(* rising edge trigger *)
IF in AND NOT edge THEN
	start := Tx;
	IF pt > t#0ms THEN Q := TRUE; END_IF;
END_IF;
edge := in;
IF q THEN
	et := Tx - start;
	IF et >= PT THEN
		Q := FALSE;
		et := t#0ms;
	END_IF;
END_IF;


(* revision history
hm	4. aug 2006		rev 1.0
	original version

hm	17. sep 2007	rev 1.1
	replaced time() with T_PLC_MS() for compatibility reasons
	
*)
END_FUNCTION_BLOCK

(* POU engineering/signal generators/pwm_pw, ST *)
FUNCTION_BLOCK pwm_pw
VAR_INPUT
	F : REAL;
	PW : TIME;
END_VAR
VAR_OUTPUT
	Q : BOOL;
END_VAR
VAR
	clk: CLK_Prg;
	pulse: TP_R;
END_VAR

(*
	version 1.1	25 feb 2007
	programmer 	oscat
	tested BY		oscat

this signal generator generates a square wave signal which is specified by the frequency and the pulse width.
*)
CLK(PT := REAL_TO_TIME(1000/F));
Pulse(in := clk.Q, pt := pw);
Q := pulse.Q;

(* revision history

hm		25. feb 2007	rev 1.1
	recoded in st for better performance and better portability

*)
END_FUNCTION_BLOCK

(* POU engineering/signal generators/rmp_soft, ST *)
FUNCTION_BLOCK rmp_soft
VAR_INPUT
	IN : BOOL;
	val : BYTE;
END_VAR
VAR_INPUT CONSTANT
	pt_on: TIME := T#100ms;
	PT_off : TIME := T#100ms;
END_VAR
VAR CONSTANT
	steps : INT := 255;
END_VAR
VAR_OUTPUT
	Out : BYTE := 0;
END_VAR
VAR
	last_step : TIME := T#0ms;
	now : TIME;
	x :REAL := 0;
END_VAR

(*
	version 1.2	17 sep 2007
	programmer 	oscat
	tested BY		oscat

this soft on/off ramp generator generates a soft on and soft off ramp while the max on value is set by the input
the time for a full ramp can be set by config variables for up and down ramp.
*)
(* read system time *)
now := DWORD_TO_TIME(T_PLC_MS());

IF in  AND out < val THEN
	(* generate on ramp *)
	x := out + TIME_TO_REAL(now -last_step)*steps/TIME_TO_REAL(pt_on);
	IF x > val THEN
		out := val;
		x := val;
	ELSE out := REAL_TO_BYTE(x); END_IF;
	last_step := now;
ELSIF NOT in AND out > 0 THEN
	(* generate off ramp *)
	x := out - TIME_TO_REAL(now - last_step)*steps/TIME_TO_REAL(pt_off);
	IF x  < 0 THEN
		out := 0;
		x := 0;
	ELSE out := REAL_TO_BYTE(x); END_IF;
	last_step := now;
ELSIF in AND out > val THEN
	(* generate ramp down to input value *)
	x := out - TIME_TO_REAL(now - last_step)*steps/TIME_TO_REAL(pt_off);
	IF x  < val THEN
		out := val;
		x := val;
	ELSE out := REAL_TO_BYTE(x); END_IF;
	last_step := now;
END_IF;
IF out = val OR out = 0 THEN last_step := now; END_IF;


(* revision history

hm 22.1.2007	rev 1.1
	deleted unused variables X1 and I, X2 and X3

hm	17.9.2007	rev 1.2
	replaced time() with t_plc_ms() for compatibility reasons

*)
END_FUNCTION_BLOCK

(* POU engineering/signal generators/rmp_W, ST *)
FUNCTION_BLOCK rmp_W
VAR_INPUT
	SET : BOOL := FALSE;
	PT : TIME;
	EN : BOOL := TRUE;
	UP : BOOL := TRUE;
	RST : BOOL := FALSE;
END_VAR
VAR_OUTPUT
	out : WORD;
	busy : BOOL;
	high : BOOL;
	low : BOOL;
END_VAR
VAR
	last_step : DWORD;
	now : DWORD;
	tmp: DWORD;
	edge: BOOL;
	N: WORD;
END_VAR

(*
	version 1.5	5. oct 2007
	programmer 	oscat
	tested BY		oscat

this ramp generator generates a Word wide ramp with 65535 steps
the generator has an asynchronous set and reset
the ramp is controlled by PT which is the total ramp time for a full sweep from 0..65535
an UD input controlls the direction Up or Down and the E input enables the ramp generation
a busy output indicates that the ramp is running, busy false means output is stable.
the outputs low and high will be true when the output has reached its max or min value.
*)
(* read system time *)
now := T_PLC_US();

(* calculate the necessary step response *)
IF pt = t#0s THEN
	tmp := 65535;
ELSE
	tmp := SHL(now - last_step, 8) / (TIME_TO_DWORD(pt)*1000);
END_IF;
IF tmp > 65535 THEN N:= 65535; ELSE N:= DWORD_TO_BYTE(tmp); END_IF;

(* detetct edge on en *)
IF en AND NOT edge THEN
	last_step := now;
(* check for asynchronous set or reset *)
ELSIF rst THEN
	out := 0;
ELSIF set  THEN
	out := 65535;
ELSIF en AND N > 0 THEN
	(* generate ramp *)
	last_step := last_step + SHR(N * TIME_TO_DWORD(pt) * 1000,16);
	IF UP THEN
		IF out > 65535 - N THEN out := 65535; ELSE out := out + N; END_IF;
	ELSE
		IF out < N THEN out := 0; ELSE out := out - N; END_IF;
	END_IF;
END_IF;
edge := en;

(* checks for outputs stable and reset or set busy flag *)
IF out = 0 THEN
	busy := FALSE;
	low := TRUE;
	high := FALSE;
ELSIF out = 65535 THEN
	busy := FALSE;
	high := TRUE;
	low := FALSE;
ELSE
	busy := en;
	high := FALSE;
	low := FALSE;
END_IF;

(* revision history:

hm 4.10.2006		rev 1.1
	added the busy output which signals that the ramp is running.

hm 22.1.2007		rev 1.2
	deleted unused variable step

hm	17.9.2007		rev 1.3
	replaced time() with t_plc_ms() for compatibility reasons

hm	28. sep 2007	rev 1.4
	added outputs on and off
	busy is now disabled while en is false
	new coding for higher accuracy and performance

hm	5. oct 2007		rev 1.5
	added statements to allow for PT to be t#0s output jumps to max or min immediately

*)
END_FUNCTION_BLOCK

(* POU engineering/signal processing/AIN, ST *)
FUNCTION AIN : REAL
VAR_INPUT
	in : DWORD;
END_VAR
VAR_INPUT CONSTANT
	Bits : BYTE;
	sign : BYTE := 255;
	low : REAL := 0;
	high : REAL := 10;
END_VAR
VAR CONSTANT
	ff : DWORD := 16#FFFFFFFF;
END_VAR
VAR
	temp1 : DWORD;
	temp2 : DWORD;
	sx : BOOL;
END_VAR

(*
version 1.3	13 sep 2007
programmer 	oscat
tested by		tobias

Ain converts signals from A/D converters or other analog sources to an internal real value
the lowest number of bits are extracted from the input word and the sign will be extracted if available separately.
the output signal is then conditioned to range from low to high values for a 0 to max value on the analog inputs:
for example a 15bit input (bits := 12) with sign at bit 15 (0..15) will deliver 0.0 (low value at 0) for an input value of 2#0000_0000_0000
an input value of 2#1111_1111_1111 will deliver 10.0 on the output (high value set to 10).

*) 
(* extract the sign bit *)
IF sign < 32 THEN
	temp1 := SHR(in,sign);
	sx := temp1.0;
ELSE
	sx := FALSE;
END_IF;
temp1 := SHR(ff,32-bits);
temp2 := in AND temp1;
AIN := (high - low)*temp2 / temp1 + low;
IF sx THEN AIN := AIN * -1; END_IF;

(* revision history
hm 18.8.2006	rev 1.1
	fixed an error with low value negative and high value 0.

hm 19.1.2007	rev 1.2
	fixed an error with sign bit.

hm	13.9.2007	rev 1.3
	changed code to avoid warning under codesys 2.8.1
*)
END_FUNCTION

(* POU engineering/signal processing/Aout, ST *)
FUNCTION Aout : DWORD
VAR_INPUT
	in : REAL;
END_VAR
VAR_INPUT CONSTANT
	Bits : BYTE;
	sign : BYTE := 255;
	low : REAL := 0;
	high : REAL := 10;
END_VAR
VAR CONSTANT
	ff : DWORD := 2#1;
END_VAR
VAR
	in2 : REAL;
	sx : BOOL;
END_VAR

(*
version 1.2	13 sep 2007
programmer 	oscat
tested by		tobias

this module conditions an internal real value for a signal output D/A converter.
Aout converts and internal real value to a word for an D/A converter or other output devices.
The input value is converted to a n-bit wide output and a sign bit is set separately as specified.
the outout min value is set for the specified min input value and the max output is set for the max input value.
an input higher or lower then the max or min value will set the respective max or min value or the output.


*) 
(* if sign bit is defined *)
IF sign < 32 THEN
	sx := sign_R(in);
	in2 := ABS(in);
ELSE
	in2 := in;
END_IF;

(* begrenze in auf die zulässigen werte *)
IF in2 < low THEN
	in2 := low;
ELSIF in2 > high THEN
	in2 := high;
END_IF;

(* Berechne den Ausgnagswert *)
Aout := REAL_TO_DWORD((in2 - low) / (high - low) * (EXPT(2,bits) -1));
IF sx THEN Aout := SHL(ff,sign) OR Aout; END_IF;

(*
revision history

hm 18.1.2007		rev 1.1
	renamed Modul to aout.
	changed Output to 32 Bit max.
	corrected error with sign bit.

hm	13.9.2007	rev 1.2
	changed code to avoid warning under codesys 2.8.1
*)
END_FUNCTION

(* POU engineering/signal processing/delay, ST *)
FUNCTION_BLOCK delay
VAR_INPUT
	in : REAL;
	N : INT;
	rst : BOOL;
END_VAR
VAR_OUTPUT
	out : REAL;
END_VAR
VAR
	buf : ARRAY[0..31] OF REAL;
	i : INT;
END_VAR

(*
version 1.2	19. jan 2007
programmer 	hugo
tested by		tobias

this function block delays input values by each programm cycle
after N+1 cycles the in value has shifted to the out.
N can be any alue from 0 .. 32
if n = 0 the input will be present on the output without a delay.
f N > 32 then the output will be delayed by 32 cycles.
any high on rst will load the buffer with in.

*)
IF N > SIZEOF(buf) / SIZEOF(in) THEN N:= 32; END_IF;
IF rst THEN
	FOR i := 0 TO 31 DO buf[i] := 0; END_FOR;
	out := in;
ELSIF N < 1 THEN out := in;
ELSE
	IF i >= N THEN i := 0; END_IF;
	out := buf[i];
	buf[i] := in;
	i := i + 1;
END_IF;

(* revision history
hm 1.10.2006	rev 1.1
	corrected error in buffer management

hm 19.1.2007	rev 1.2
	changed reset to load the value of in instead of 0

*)
END_FUNCTION_BLOCK

(* POU engineering/signal processing/delay_4, ST *)
FUNCTION_BLOCK delay_4
VAR_INPUT
	in : REAL;
END_VAR
VAR_OUTPUT
	out1 : REAL;
	out2 : REAL;
	out3 : REAL;
	out4 : REAL;
END_VAR
VAR
	temp: REAL;
END_VAR

(*
version 1.1	19 jan 2007
programmer 	hugo
tested by		tobias

this function block delays input values by each programm cycle
after 4 cycles the in value has shifted to the out 4 and will be discarded after the next cycle
the blocks can be cascaded.

*)
out4 := out3;
out3 := out2;
out2 := out1;
out1 := temp;
temp := in;

(* revision history

hm 19.1.2007	rev 1.1
	added variable temp to add 1 delay  for q1

*)
END_FUNCTION_BLOCK

(* POU engineering/signal processing/MIX, ST *)
FUNCTION MIX : REAL
VAR_INPUT
	A, B : REAL;
	M : REAL;
END_VAR
VAR
END_VAR

(*
version 1.0	19 nov 2007
programmer 	hugo
tested by		tobias

MIX is an analog Mixer. The Output is (1-M)*A + M*B.

*)
MIX := (1-M)*A + M*B;

(* revision history
hm	19. Nov 2007		rev 1.0
	original version
*)
END_FUNCTION

(* POU engineering/signal processing/MUX_R2, ST *)
FUNCTION MUX_R2 : REAL
VAR_INPUT
	IN0 : REAL;
	IN1 : REAL;
	A : BOOL;
END_VAR
VAR
END_VAR

(*
version 1.0	19 jan 2007
programmer 	oscat
tested by		tobias

MUX_R2 is an analog Multiplexer.
one of 2 real inputs are selected and put through to out.
The Adress input A selects between 2 Real inputs IN0 and IN1, A=0 > In0, A=1 > in1.

*)
IF NOT A THEN
	MUX_R2 := IN0;
ELSE
	MUX_R2 := IN1;
END_IF;
END_FUNCTION

(* POU engineering/signal processing/MUX_R4, ST *)
FUNCTION MUX_R4 : REAL
VAR_INPUT
	IN0 : REAL;
	IN1 : REAL;
	IN2 : REAL;
	IN3 : REAL;
	A0 : BOOL;
	A1 : BOOL;
END_VAR
VAR
END_VAR

(*
version 1.0	19 jan 2007
programmer 	oscat
tested by		tobias

MUX_R4 is an analog Multiplexer.
one of 4 real inputs are selected and put through to out.
The Adress input A0 and A1 selects between the 4 Real inputs IN0.. IN1.

*)
IF NOT A0 AND NOT A1 THEN
	MUX_R4 := IN0;
ELSIF A0 AND NOT a1 THEN
	MUX_R4 := IN1;
ELSIF NOT A0 AND A1 THEN
	MUX_R4 := IN2;
ELSE
	MUX_R4 := IN3;
END_IF;
END_FUNCTION

(* POU engineering/signal processing/Offset2, ST *)
FUNCTION Offset2 : REAL
VAR_INPUT
	X : REAL;
	O1, O2, O3, O4 : BOOL;
	D : BOOL;
END_VAR
VAR_INPUT CONSTANT
	Offset_1 : REAL;
	Offset_2 : REAL;
	Offset_3 : REAL;
	Offset_4 : REAL;
	default : REAL;
END_VAR

(*
version 1.0	12 jan 2007
programmer 	oscat
tested by		tobias

The Function offset adds offsets to an analog signal depending on digital inputs.
one offset can be added at the same time, if more then one input is true, the one with the highest number (o1 .. o4) will be used.
The input D will select a default value instead of X for input.

*) 
IF D THEN Offset2 := default; ELSE Offset2 := X; END_IF;
IF O4 THEN Offset2 := Offset2 + offset_4;
ELSIF O3 THEN Offset2 := Offset2 + offset_3;
ELSIF O2 THEN Offset2 := Offset2 + offset_2;
ELSIF O1 THEN Offset2 := Offset2 + offset_1;
END_IF;
END_FUNCTION

(* POU engineering/signal processing/Override, ST *)
FUNCTION Override : REAL
VAR_INPUT
	X1, X2, X3 : REAL;
	E1 : BOOL;
	E2 : BOOL;
	E3 : BOOL;
END_VAR
VAR
END_VAR

(*
version 1.0	4 nov 2007
programmer 	oscat
tested by	tobias

MAXR deliveres the maximum absolute value of the 3 inputs X1, X2 and X3.
with the inputs E1, E2 and E3 each of the 3 inputs can be turned on or off, while the default for these 3 inputs is true.

*) 
IF E1 THEN Override := X1; END_IF;
IF E2 AND ABS(x2) > ABS(Override) THEN Override := X2; END_IF;
IF E3 AND ABS(x3) > ABS(Override) THEN Override := X3; END_IF;

(* revision history
hm		4.11.2007		rev 1.0
	original version

*)
END_FUNCTION

(* POU engineering/signal processing/scale_B2, ST *)
FUNCTION scale_B2 : REAL
VAR_INPUT
	in1: BYTE;
	in2: BYTE;
	K : REAL := 1;
	O : REAL := 0;
END_VAR
VAR_INPUT CONSTANT
	in1_min: REAL := 0;
	in1_max: REAL := 1000;
	in2_min: REAL := 0;
	in2_max: REAL := 1000;
END_VAR

(*
version 1.1	19 jan 2007
programmer 	hugo
tested by		tobias

	this functiob block can scale up to two inputs.
	the inputs have their min value at 0 and their max value at 255 while the min and max value can be either positive or negative.
	the inputs ramp between min and max values for the respective inputs to be between (0..255).
	the summed output is then scaled by an scale input K and a offset O can be added to the output.
	the min and max input configurations can be edited in the cfc editor by double clicking the symbol body.

*)
scale_B2 := 	((in1_max - in1_min)* in1 / 255 + in1_min +
				(in2_max - in2_min)* in2 / 255 + in2_min)
				* K + O;

(* revision History
hm 19.1.2007	rev 1.1
	changed outputs to real to avoid overflow of integer
	added offset for better cascading of scale functions
	changed from FB to function
*)
END_FUNCTION

(* POU engineering/signal processing/scale_B4, ST *)
FUNCTION scale_B4 : REAL
VAR_INPUT
	in1: BYTE;
	in2: BYTE;
	in3: BYTE;
	in4: BYTE;
	K : REAL := 1;
	O : REAL := 0;
END_VAR
VAR_INPUT CONSTANT
	in1_min: REAL := 0;
	in1_max: REAL := 1000;
	in2_min: REAL := 0;
	in2_max: REAL := 1000;
	in3_min: REAL := 0;
	in3_max: REAL := 1000;
	in4_min: REAL := 0;
	in4_max: REAL := 1000;
END_VAR

(*
version 1.1	19 jan 2007
programmer 	hugo
tested by		tobias

	this functiob block can scale up to 4 inputs.
	the inputs have their min value at 0 and their max value at 255 while the min and max value can be either positive or negative.
	the inputs ramp between min and max values for the respective inputs to be between (0..255).
	the summed output is then scaled by an scale input K and a offset O can be added to the output.
	the min and max input configurations can be edited in the cfc editor by double clicking the symbol body.

*)
scale_B4 := 	((in1_max - in1_min)* in1 / 255 + in1_min +
				(in2_max - in2_min)* in2 / 255 + in2_min +
				(in3_max - in3_min)* in3 / 255 + in3_min +
				(in4_max - in4_min)* in4 / 255 + in4_min)
				* K + O;

(* revision History
hm 19.1.2007	rev 1.1
	changed outputs to real to avoid overflow of integer
	added offset for better cascading of scale functions
	changed from fb to function
*)
END_FUNCTION

(* POU engineering/signal processing/scale_B8, ST *)
FUNCTION scale_B8 : REAL
VAR_INPUT
	in1: BYTE;
	in2: BYTE;
	in3: BYTE;
	in4: BYTE;
	in5: BYTE;
	in6: BYTE;
	in7: BYTE;
	in8: BYTE;
	K : REAL := 1;
	O : REAL := 0;
END_VAR
VAR_INPUT CONSTANT
	in1_min: REAL := 0;
	in1_max: REAL := 1000;
	in2_min: REAL := 0;
	in2_max: REAL := 1000;
	in3_min: REAL := 0;
	in3_max: REAL := 1000;
	in4_min: REAL := 0;
	in4_max: REAL := 1000;
	in5_min: REAL := 0;
	in5_max: REAL := 1000;
	in6_min: REAL := 0;
	in6_max: REAL := 1000;
	in7_min: REAL := 0;
	in7_max: REAL := 1000;
	in8_min: REAL := 0;
	in8_max: REAL := 1000;
END_VAR

(*
version 1.1	19 jan 2007
programmer 	hugo
tested by		tobias

	this functiob block can scale up to 8 inputs.
	the inputs have their min value at 0 and their max value at 255 while the min and max value can be either positive or negative.
	the inputs ramp between min and max values for the respective inputs to be between (0..255).
	the summed output is then scaled by an scale input K and a offset O can be added to the output.
	the min and max input configurations can be edited in the cfc editor by double clicking the symbol body.

*)
scale_B8 := 	((in1_max - in1_min)* in1 / 255 + in1_min +
				(in2_max - in2_min)* in2 / 255 + in2_min +
				(in3_max - in3_min)* in3 / 255 + in3_min +
				(in4_max - in4_min)* in4 / 255 + in4_min +
				(in5_max - in5_min)* in5 / 255 + in5_min +
				(in6_max - in6_min)* in6 / 255 + in6_min +
				(in7_max - in7_min)* in7 / 255 + in7_min +
				(in8_max - in8_min)* in8 / 255 + in8_min)
				* K + O;

(* revision History
hm 19.1.2007	rev 1.1
	changed outputs to real to avoid overflow of integer
	added offset for better cascading of scale functions
*)
END_FUNCTION

(* POU engineering/signal processing/scale_X2, ST *)
FUNCTION scale_X2 : REAL
VAR_INPUT
	in1: BOOL;
	in2: BOOL;
	K : REAL := 1;
	O : REAL := 0;
END_VAR
VAR_INPUT CONSTANT
	in1_min: REAL := 0;
	in1_max: REAL := 1000;
	in2_min: REAL := 0;
	in2_max: REAL := 1000;
END_VAR

(*
version 1.0	19 jan 2007
programmer 	hugo
tested by		tobias

	this functiob block can scale up to two inputs.
	the input can select between two values with true or false.
	the summed output is then scaled by an scale input K and a offset O can be added to the output.
	the min and max input configurations can be edited in the cfc editor by double clicking the symbol body.

*)
IF NOT in1 THEN scale_x2 := in1_min; ELSE scale_x2 := in1_max; END_IF;
IF NOT in2 THEN scale_x2 := scale_x2 + in2_min; ELSE scale_x2 := scale_x2 + in2_max; END_IF;
scale_X2 := scale_X2 * k + O;

(* revision history

*)
END_FUNCTION

(* POU engineering/signal processing/scale_X4, ST *)
FUNCTION scale_X4 : REAL
VAR_INPUT
	in1: BOOL;
	in2: BOOL;
	in3: BOOL;
	in4: BOOL;
	K : REAL := 1;
	O : REAL := 0;
END_VAR
VAR_INPUT CONSTANT
	in1_min: REAL := 0;
	in1_max: REAL := 1000;
	in2_min: REAL := 0;
	in2_max: REAL := 1000;
	in3_min: REAL := 0;
	in3_max: REAL := 1000;
	in4_min: REAL := 0;
	in4_max: REAL := 1000;
END_VAR

(*
version 1.0	19 jan 2007
programmer 	hugo
tested by		tobias

	this function can scale up to 4 inputs.
	the input can select between two values with true or false.
	the summed output is then scaled by an scale input K and a offset O can be added to the output.
	the min and max input configurations can be edited in the cfc editor by double clicking the symbol body.

*)
IF NOT in1 THEN scale_X4 := in1_min; ELSE scale_X4 := in1_max; END_IF;
IF NOT in2 THEN scale_x4 := scale_x4 + in2_min; ELSE scale_x4 := scale_x4 + in2_max; END_IF;
IF NOT in3 THEN scale_x4 := scale_x4 + in3_min; ELSE scale_x4 := scale_x4 + in3_max; END_IF;
IF NOT in4 THEN scale_x4 := scale_x4 + in4_min; ELSE scale_x4 := scale_x4 + in4_max; END_IF;
scale_X4 := scale_X4 * k + O;

(* revision history

*)
END_FUNCTION

(* POU engineering/signal processing/scale_X8, ST *)
FUNCTION scale_X8 : REAL
VAR_INPUT
	in1: BOOL;
	in2: BOOL;
	in3: BOOL;
	in4: BOOL;
	in5: BOOL;
	in6: BOOL;
	in7: BOOL;
	in8: BOOL;
	K : REAL := 1;
	O : REAL := 0;
END_VAR
VAR_INPUT CONSTANT
	in1_min: REAL := 0;
	in1_max: REAL := 1000;
	in2_min: REAL := 0;
	in2_max: REAL := 1000;
	in3_min: REAL := 0;
	in3_max: REAL := 1000;
	in4_min: REAL := 0;
	in4_max: REAL := 1000;
	in5_min: REAL := 0;
	in5_max: REAL := 1000;
	in6_min: REAL := 0;
	in6_max: REAL := 1000;
	in7_min: REAL := 0;
	in7_max: REAL := 1000;
	in8_min: REAL := 0;
	in8_max: REAL := 1000;
END_VAR

(*
version 1.0	19 jan 2007
programmer 	hugo
tested by		tobias

	this function can scale up to 4 inputs.
	the input can select between two values with true or false.
	the summed output is then scaled by an scale input K and a offset O can be added to the output.
	the min and max input configurations can be edited in the cfc editor by double clicking the symbol body.

*)
IF NOT in1 THEN scale_x8 := in1_min; ELSE scale_x8 := in1_max; END_IF;
IF NOT in2 THEN scale_x8 := scale_x8 + in2_min; ELSE scale_x8 := scale_x8 + in2_max; END_IF;
IF NOT in3 THEN scale_x8 := scale_x8 + in3_min; ELSE scale_x8 := scale_x8 + in3_max; END_IF;
IF NOT in4 THEN scale_x8 := scale_x8 + in4_min; ELSE scale_x8 := scale_x8 + in4_max; END_IF;
IF NOT in5 THEN scale_x8 := scale_x8 + in5_min; ELSE scale_x8 := scale_x8 + in5_max; END_IF;
IF NOT in6 THEN scale_x8 := scale_x8 + in6_min; ELSE scale_x8 := scale_x8 + in6_max; END_IF;
IF NOT in7 THEN scale_x8 := scale_x8 + in7_min; ELSE scale_x8 := scale_x8 + in7_max; END_IF;
IF NOT in8 THEN scale_x8 := scale_x8 + in8_min; ELSE scale_x8 := scale_x8 + in8_max; END_IF;
scale_X8 := scale_X8 * k + O;

(* revision history

*)
END_FUNCTION

(* POU engineering/signal processing/SH, ST *)
FUNCTION_BLOCK SH
VAR_INPUT
	in : REAL;
	CLK : BOOL;
END_VAR
VAR_OUTPUT
	out : REAL;
	trig : BOOL;
END_VAR
VAR
	edge : BOOL;
END_VAR

(*
version 1.1	16 jan 2007
programmer 	hugo
tested by		tobias

this sample and hold module samples an input at the rising edge of clk an stores it in out.
the out stays stable until the next rising clk edge appears.
a trigger output as active for one cycle when the output was updated.

*)
IF clk AND NOT edge THEN
	out := in;
	trig := TRUE;
ELSE;
	trig := FALSE;
END_IF;
edge := clk;

(* revision history

hm 16.1.2007	rev 1.1
	added trig output

*)
END_FUNCTION_BLOCK

(* POU engineering/signal processing/SH_1, ST *)
FUNCTION_BLOCK SH_1
VAR_INPUT
	in : REAL;
	PT : TIME;
END_VAR
VAR_OUTPUT
	out : REAL;
	Trig : BOOL;
END_VAR
VAR
	last : TIME;
	tx: TIME;
END_VAR

(*
version 1.2	17 sep 2007
programmer 	hugo
tested by		tobias

this sample and hold module samples an input every PT seconds.
after a ample is taken the output Trig will be active for one cycle.

*)
(* read system time *)
tx := DWORD_TO_TIME(T_PLC_MS());

IF tx - last >= PT THEN
	last := tx;
	out := in;
	trig := TRUE;
ELSE
	trig := FALSE;
END_IF;

(* revision history

HM	6.1.2007	rev 1.1
	added trig output

HM	17.9.2007	rev 1.2
	replaced time() with T_PLC_MS() for compatibility reasons
*)
END_FUNCTION_BLOCK

(* POU engineering/signal processing/SH_2, ST *)
FUNCTION_BLOCK SH_2
VAR_INPUT
	in : REAL;
	PT : TIME;
	N : INT;
	disc : INT;
END_VAR
VAR_OUTPUT
	out : REAL;
	trig : BOOL;
	avg : REAL;
	high: REAL;
	low: REAL;
END_VAR
VAR
	M : INT;
	buf : ARRAY[0..15] OF REAL;
	buf2 : ARRAY[0..15] OF REAL;
	last : TIME;
	i : INT;
	start: INT;
	temp: REAL;
	stop: INT;
	tx: TIME;
END_VAR

(*
version 1.3	17 sep 2007
programmer 	hugo
tested by		tobias

this sample and hold module samples an input every PT seconds.
this sample and hold also does avg and other calculations with the input data.
an average is calculated over N samples while for this calculation disc samples are discarded,
disc = 0 all samples are averaged,
if disc = 1 the lowest value is ignored,
if disc = 2 the lowest and highest values are ignored, 
and so on.....

*)
(* read system time *)
tx := DWORD_TO_TIME(T_PLC_MS());

IF tx - last >= PT THEN
	last := tx;
	trig := TRUE;

	(* limit M to 0..16 *)
	M := LIMIT(1,N,16);

	(* edge detected lets take the sample *)
	FOR i := M - 1 TO 1 BY -1 DO buf2[i] := buf2[i-1]; END_FOR;
	buf2[0] := in;
	out := in;
	buf := buf2;

	(* sort the ARRAY lowest value AT 0 *)
	FOR start := 0 TO M - 2 DO
		FOR i := start+1 TO M - 1 DO
			IF buf[start] > buf[i] THEN
				temp := buf[start];
				buf[start] := buf[i];
				buf[i] := temp;
			END_IF;
		END_FOR;
	END_FOR;

	(* any calculation with the samples is here *)
	stop := M - 1 - disc / 2;
	start := 0 + disc / 2;
	IF NOT even(disc) THEN start := start + 1; END_IF;
	avg := 0;
	FOR i := start TO stop DO avg := avg + buf[i]; END_FOR;
	avg := avg / (stop - start +1);
	low := buf[start];
	high := buf[stop];
ELSE
	Trig := FALSE;
END_IF;

(* revision history
hm 20.1.2007	rev 1.1
	added input N to specify the amout of samples for average and high low calculations
	added trig output

hm 10.9.2007 rev 1.2
	an error would be generated if N was set to 0, now n is forced to1 if set to 0.
	index was out of array.

hm	17.9.2007	rev 1.3
	replaced time() with t_plc_ms() for compatibility reasons

*)
END_FUNCTION_BLOCK

(* POU mathematical/even, ST *)
FUNCTION even : BOOL
VAR_INPUT
	in : INT;
END_VAR
VAR
END_VAR


(*
version 1.0	1 oct 2006
programmer 	hugo
tested by		tobias

this function chacks an input for even  value
the output is true if the input is even.
execution time on wago 750 - 841 =  10  us
*)
IF (in MOD 2) = 0 THEN  even := TRUE; ELSE even := FALSE; END_IF;
END_FUNCTION

(* POU engineering/signal processing/SH_T, ST *)
FUNCTION_BLOCK SH_T
VAR_INPUT
	in : REAL;
	EN : BOOL;
END_VAR
VAR_OUTPUT
	out : REAL;
END_VAR
VAR
END_VAR

(*
version 1.0	1 sep 2006
programmer 	hugo
tested by		tobias

this sample and hold module samples an input while en is high.
during the high time of en the output follows in.
the out stays stable until the en goes high again.
*)
IF en THEN out := in; END_IF;
END_FUNCTION_BLOCK

(* POU engineering/signal processing/stair, ST *)
FUNCTION stair : REAL
VAR_INPUT
	X : REAL;
	D : REAL;
END_VAR
VAR
	temp: REAL;
END_VAR


(*
version 1.0	28 jan 2007
programmer 	oscat
tested by		tobias

the function stair converts an anlog input signal to a staircase like output.
D is the step width for the output signal.
if D = 0 then the output follows the input without a chage.
*) 
temp := modR(X, D);
IF ABS(temp) < D / 2 THEN
	IF X > 0 THEN stair := X - temp; ELSE stair := X - temp; END_IF;
ELSE
	IF X > 0 THEN stair := X - temp + D; ELSE stair := X - temp - D; END_IF;
END_IF;
END_FUNCTION

(* POU engineering/signal processing/stair2, ST *)
FUNCTION_BLOCK stair2
VAR_INPUT
	X : REAL;
	D : REAL;
END_VAR
VAR_OUTPUT
	Y: REAL;
END_VAR
VAR_TEMP
	tmp : REAL;
END_VAR


(*
version 1.0	28 jan 2007
programmer 	oscat
tested by		tobias

the function stair2 converts an anlog input signal to a staircase like output.
D is the step width for the output signal. the output will use D as a hysteresis for a stairchange.
if D = 0 then the output follows the input without a chage.
*) 
tmp := TRUNC(X / D);

IF X >= Y AND X >= 0 THEN
	Y := TRUNC(X / D) * D;
ELSIF X < Y AND X >= 0 THEN
	Y := (TRUNC(X/d) + 1) * D;
ELSIF X >= Y AND X < 0 THEN
	Y := (TRUNC(X/D)-1) * D;
ELSIF X < Y AND X < 0 THEN
	Y := TRUNC(X/D) *D;
END_IF;
END_FUNCTION_BLOCK

(* POU Logic/FF edge triggered/FF_D2E, ST *)
FUNCTION_BLOCK FF_D2E
VAR_INPUT
	D0 : BOOL := 0;
	D1 : BOOL := 0;
	CLK : BOOL;
	RST : BOOL := 0;
END_VAR
VAR_OUTPUT
	Q0 : BOOL := 0;
	Q1 : BOOL := 0;
END_VAR
VAR
	edge : BOOL;
END_VAR

(*
version 1.0	4 aug 2006
programmer 	hugo
tested by		tobias

dual D-type flip flop with reset and rising clock trigger

executioin TIME on wago 750-841 = 6us
*)
IF rst THEN
	Q0 := FALSE;
	Q1 := FALSE;
ELSE
	IF clk AND NOT edge THEN
		Q0 := D0;
		Q1 := D1;
	END_IF;
END_IF;
edge := CLK;
END_FUNCTION_BLOCK

(* POU Logic/FF edge triggered/FF_D4E, ST *)
FUNCTION_BLOCK FF_D4E
VAR_INPUT
	D0 : BOOL := 0;
	D1 : BOOL := 0;
	D2 : BOOL := 0;
	D3 : BOOL := 0;
	CLK : BOOL;
	RST : BOOL := 0;
END_VAR
VAR_OUTPUT
	Q0 : BOOL := 0;
	Q1 : BOOL := 0;
	Q2 : BOOL := 0;
	Q3 : BOOL := 0;
END_VAR
VAR
	edge : BOOL;
END_VAR


(*
version 1.0	4 aug 2006
programmer 	hugo
tested by		tobias

quad D-type flip flop with reset and rising clock trigger

executioin TIME on wago 750-841 = 6us
*)
IF rst THEN
	Q0 := FALSE;
	Q1 := FALSE;
	Q2 := FALSE;
	Q3 := FALSE;
ELSE
	IF clk AND NOT edge THEN
		Q0 := D0;
		Q1 := D1;
		Q2 := D2;
		Q3 := D3;
	END_IF;
END_IF;
edge := CLK;
END_FUNCTION_BLOCK

(* POU Logic/FF edge triggered/FF_DRE, ST *)
FUNCTION_BLOCK FF_DRE
VAR_INPUT
	SET : BOOL;
	D : BOOL;
	CLK : BOOL;
	RST : BOOL;
END_VAR
VAR_OUTPUT
	Q : BOOL := 0;
END_VAR
VAR
	edge : BOOL;
END_VAR


(*
version 1.0	4 aug 2006
programmer 	hugo
tested by		tobias

D-type flip flop with set, reset and rising clock trigger
executioin TIME on wago 750-841 = 8us
*)
IF rst THEN
	Q := FALSE;
ELSIF set AND NOT rst THEN
	Q := TRUE;
ELSE
	IF clk AND NOT edge THEN Q := D; END_IF;
END_IF;
edge := CLK;
END_FUNCTION_BLOCK

(* POU Logic/FF edge triggered/FF_JKE, ST *)
FUNCTION_BLOCK FF_JKE
VAR_INPUT
	SET : BOOL;
	J : BOOL;
	CLK : BOOL;
	K : BOOL;
	RST : BOOL;
END_VAR
VAR_OUTPUT
	Q : BOOL := 0;
END_VAR
VAR
	edge : BOOL;
END_VAR


(*
version 1.0	4 aug 2006
programmer 	hugo
tested by		tobias

JK-type flip flop with set, reset and rising clock trigger
set and reset are asynchron while the FF is rising edge triggered
J=0 and K=0 and CLK >>> no action
J=1 and K=0 and CLK >>> output = 1
J=0 and K=1 and CLK >>> output = 0
J=1 and K=1 and CLK >>> toggle output

executioin TIME on wago 750-841 = 8us
*)
IF rst THEN
	Q := FALSE;
ELSIF set AND NOT rst THEN
	Q := TRUE;
ELSE
	IF clk AND NOT edge THEN
		IF J AND NOT K THEN Q := TRUE;
		ELSIF K AND NOT J THEN Q := FALSE;
		ELSIF K AND J THEN Q:= NOT Q;
		END_IF;
	END_IF;
END_IF;
edge := CLK;
END_FUNCTION_BLOCK

(* POU Logic/FF edge triggered/SHR_4E, ST *)
FUNCTION_BLOCK SHR_4E
VAR_INPUT
	SET : BOOL :=0;
	D0: BOOL := 0;
	CLK: BOOL;
	RST: BOOL :=0;
END_VAR
VAR_OUTPUT
	Q0: BOOL :=0;
	Q1: BOOL :=0;
	Q2: BOOL :=0;
	Q3: BOOL :=0;
END_VAR
VAR
	edge : BOOL :=1;
END_VAR

(*
version 1.0	4 aug 2006
programmer 	hugo
tested by		tobias

4 bit shift register with reset

executioin TIME on wago 750-841 =  8 us
*)
(* flankenerkennung clk wird high und edge war high reset ist nicht aktiv und set ist nicht aktiv *)
IF CLK AND edge AND NOT rst AND NOT set THEN
	edge := FALSE;	(* flanke wurde erkannt und weitere flankenerkennung wird verhindert bis edge wieder true ist *)
	(* hier ist der code für das ff aktivity *)
	Q3 := Q2;
	Q2 := Q1;
	Q1 := Q0;
	Q0 := D0;
END_IF
IF NOT clk THEN edge := TRUE; END_IF;	(* sobald clk wieder low wird warten auf nächste flanke *)
IF set AND NOT rst THEN						(* ausgang asynchron setzen wenn set aktiv und reset inaktiv. reset hat immer vorrang *)
	Q0 := TRUE;
	Q1 := TRUE;
	Q2 := TRUE;
	Q3 := TRUE;
END_IF;
IF rst THEN									(* wenn reset aktiv dann ausgang rücksetzen *)
	Q0 := FALSE;
	Q1 := FALSE;
	Q2 := FALSE;
	Q3 := FALSE;
END_IF;
END_FUNCTION_BLOCK

(* POU Logic/FF edge triggered/SHR_4UDE, ST *)
FUNCTION_BLOCK SHR_4UDE
VAR_INPUT
	set : BOOL :=0;
	D0: BOOL := 0;
	D3: BOOL := 0;
	CLK: BOOL;
	DN : BOOL :=0;
	RST: BOOL :=0;

END_VAR
VAR_OUTPUT
	Q0: BOOL :=0;
	Q1: BOOL :=0;
	Q2: BOOL :=0;
	Q3: BOOL :=0;
END_VAR
VAR
	edge : BOOL :=1;
END_VAR

(*
version 1.0	4 aug 2006
programmer 	hugo
tested by		tobias

4 bit shift register with reset up / down direction input

executioin TIME on wago 750-841 =  8 us
*)
(* flankenerkennung clk wird high und edge war high reset ist nicht aktiv und set ist nicht aktiv *)
IF CLK AND edge AND NOT rst AND NOT set THEN
	edge := FALSE;	(* flanke wurde erkannt und weitere flankenerkennung wird verhindert bis edge wieder true ist *)
	(* hier ist der code für das ff aktivity *)
	IF NOT dn THEN
		Q3 := Q2;
		Q2 := Q1;
		Q1 := Q0;
		Q0 := D0;
	ELSE
		Q0 := Q1;
		Q1 := Q2;
		Q2 := Q3;
		Q3 := D3;
	END_IF
END_IF
IF NOT clk THEN edge := TRUE; END_IF;	(* sobald clk wieder low wird warten auf nächste flanke *)
IF set AND NOT rst THEN						(* ausgang asynchron setzen wenn set aktiv und reset inaktiv. reset hat immer vorrang *)
	Q0 := TRUE;
	Q1 := TRUE;
	Q2 := TRUE;
	Q3 := TRUE;
END_IF;
IF rst THEN									(* wenn reset aktiv dann ausgang rücksetzen *)
	Q0 := FALSE;
	Q1 := FALSE;
	Q2 := FALSE;
	Q3 := FALSE;
END_IF;
END_FUNCTION_BLOCK

(* POU Logic/FF edge triggered/SHR_8PLE, ST *)
FUNCTION_BLOCK SHR_8PLE
VAR_INPUT
	Din : BOOL;
	Dload : BYTE;
	CLK: BOOL;
	UP: BOOL :=1;
	load : BOOL :=0;
	RST: BOOL :=0;
END_VAR
VAR_OUTPUT
	DOut: BOOL :=0;
END_VAR
VAR
	edge : BOOL :=1;
	register : BYTE := 0;
END_VAR

(*
version 1.0	4 aug 2006
programmer 	hugo
tested by		tobias

8 bit shift register with reset and parallel load
the register can shift up or down
it also has a serial input.
the Din input is on Bit0 for up shift and on bit 7 for down shift
the Dout output is on Bit7 for up shift and on bit 0 for down shift
paralle clock is performed clock synchron while a shift is performed first and then the register is reloaded

executioin TIME on wago 750-841 =  6 us
*)
(* flankenerkennung clk wird high und edge war high reset ist nicht aktiv und set ist nicht aktiv *)
IF CLK AND edge AND NOT rst THEN
	edge := FALSE;	(* flanke wurde erkannt und weitere flankenerkennung wird verhindert bis edge wieder true ist *)
	(* hier ist der code für das flankenevent *)
	IF UP THEN						(*shift up *)
		register := SHL(register,1);
		register.0 := Din;
		Dout := register.7;
	ELSE								(* shift down *);
		register := SHR(register,1);
		register.7 := Din;
		Dout := register.0;
	END_IF;
	IF load THEN							(* the byte on Din will be loaded if load = true *)
		register := Dload;
		IF up THEN Dout := register.7; ELSE Dout := register.0; END_IF;
	END_IF;
END_IF;
IF NOT clk THEN edge := TRUE; END_IF;	(* sobald clk wieder low wird warten auf nächste flanke *)
IF rst THEN									(* wenn reset aktiv dann ausgang rücksetzen *)
	register := 0;
	Dout := FALSE;
END_IF;
END_FUNCTION_BLOCK

(* POU Logic/FF edge triggered/SHR_8UDE, ST *)
FUNCTION_BLOCK SHR_8UDE
VAR_INPUT
	set : BOOL :=0;
	D0: BOOL := 0;
	D7: BOOL := 0;
	CLK: BOOL;
	DN : BOOL :=0;
	RST: BOOL :=0;
END_VAR
VAR_OUTPUT
	Q0: BOOL :=0;
	Q1: BOOL :=0;
	Q2: BOOL :=0;
	Q3: BOOL :=0;
	Q4: BOOL :=0;
	Q5: BOOL :=0;
	Q6: BOOL :=0;
	Q7: BOOL :=0;
END_VAR
VAR
	edge : BOOL :=1;
END_VAR

(*
version 1.0	4 aug 2006
programmer 	hugo
tested by		tobias

8 bit shift register with reset

executioin TIME on wago 750-841 =  8 us
*)
(* flankenerkennung clk wird high und edge war high reset ist nicht aktiv und set ist nicht aktiv *)
IF CLK AND edge AND NOT rst AND NOT set THEN
	edge := FALSE;	(* flanke wurde erkannt und weitere flankenerkennung wird verhindert bis edge wieder true ist *)
	(* hier ist der code für das ff aktivity *)
	IF NOT dn THEN
		Q7 := Q6;
		Q6 := Q5;
		Q5 := Q4;
		Q4 := Q3;
		Q3 := Q2;
		Q2 := Q1;
		Q1 := Q0;
		Q0 := D0;
	ELSE
		Q0 := Q1;
		Q1 := Q2;
		Q2 := Q3;
		Q3 := Q4;
		Q4 := Q5;
		Q5 := Q6;
		Q6 := Q7;
		Q7 := D7;
	END_IF
END_IF
IF NOT clk THEN edge := TRUE; END_IF;	(* sobald clk wieder low wird warten auf nächste flanke *)
IF set AND NOT rst THEN						(* ausgang asynchron setzen wenn set aktiv und reset inaktiv. reset hat immer vorrang *)
	Q0 := TRUE;
	Q1 := TRUE;
	Q2 := TRUE;
	Q3 := TRUE;
	Q4 := TRUE;
	Q5 := TRUE;
	Q6 := TRUE;
	Q7 := TRUE;
END_IF;
IF rst THEN									(* wenn reset aktiv dann ausgang rücksetzen *)
	Q0 := FALSE;
	Q1 := FALSE;
	Q2 := FALSE;
	Q3 := FALSE;
	Q4 := FALSE;
	Q5 := FALSE;
	Q6 := FALSE;
	Q7 := FALSE;
END_IF;
END_FUNCTION_BLOCK

(* POU Logic/FF pulse triggered/LTCH, ST *)
FUNCTION_BLOCK LTCH
VAR_INPUT
	D : BOOL;
	L : BOOL;
	RST : BOOL := 0;
END_VAR
VAR_OUTPUT
	Q : BOOL := 0;
END_VAR
VAR
END_VAR

(*
version 1.0	4 aug 2006
programmer 	hugo
tested by		tobias

Transparent Latch with asynchronous reset

executioin TIME on wago 750-841 = 5us
*)
(* as long as L is true, the latch is transparent and and change of D is transferred to Q *)
(* of course only when there is no asynchronous reset *)
IF L AND NOT rst THEN Q := D;	(* latch is transparent *)
ELSIF rst THEN Q:= 0;			(* if asynchronous reset then Q=0 *)
END_IF;
END_FUNCTION_BLOCK

(* POU Logic/FF pulse triggered/LTCH_4, ST *)
FUNCTION_BLOCK LTCH_4
VAR_INPUT
	D0 : BOOL;
	D1 : BOOL;
	D2 : BOOL;
	D3 : BOOL;
	L : BOOL;
	RST : BOOL := 0;
END_VAR
VAR_OUTPUT
	Q0 : BOOL := 0;
	Q1 : BOOL := 0;
	Q2 : BOOL := 0;
	Q3 : BOOL := 0;
END_VAR
VAR
END_VAR

(*
version 1.0	4 aug 2006
programmer 	hugo
tested by		tobias

Quad Transparent Latch with asynchronous reset

executioin TIME on wago 750-841 = 5us
*)
(* as long as L is true, the latch is transparent and and change of D is transferred to Q *)
(* of course only when there is no asynchronous reset *)
IF L AND NOT rst THEN
	Q0 := D0;	(* latch is transparent *)
	Q1 := D1;
	Q2 := D2;
	Q3 := D3;
ELSIF rst THEN
	Q0 := FALSE;			(* if asynchronous reset then Q=0 *)
	Q1 := FALSE;
	Q2 := FALSE;
	Q3 := FALSE;
END_IF;
END_FUNCTION_BLOCK

(* POU Logic/gate logic/Bit_Count, ST *)
FUNCTION Bit_Count : INT
VAR_INPUT
	IN : DWORD;
END_VAR
VAR
END_VAR

(*
version 1.1	10 sep 2007
programmer 	hugo
tested by		tobias

BIT_COUNT counts the amount True of bits in a dword.
for exabple: bit_count(3) returns 2 because two bits (bits 0 and 1) are true and all others are false. 

*)
WHILE in > 0 DO
	IF in.0 THEN Bit_Count := Bit_Count +1; END_IF;
	in := SHR(in,1);
END_WHILE;

(* revision history
5.7.2007	rev 1.0		original version

10.9.2007	rev 1.1		hm
	changed algorithm for better performace
	the execution time has reduced by a factor of 5
	deleted unused variable temp
*)
END_FUNCTION

(* POU Logic/gate logic/Bit_of_Dword, ST *)
FUNCTION Bit_of_Dword : BOOL
VAR_INPUT
	in : DWORD;
	N : BYTE;
END_VAR
VAR
	temp: DWORD;
END_VAR

(*
version 1.0	4 aug 2006
programmer 	hugo
tested by		tobias

this function extracts a single bit from the nth position from right (right is lowest bit)
the lowest Bit (Bit0 from in) is selected with N=0.
 *)
temp := SHR(in,n);
Bit_of_Dword := temp.0;
END_FUNCTION

(* POU Logic/gate logic/Byte_of_bit, ST *)
FUNCTION Byte_of_bit : BYTE
VAR_INPUT
	B0:BOOL;
	B1:BOOL;
	B2:BOOL;
	B3:BOOL;
	B4:BOOL;
	B5:BOOL;
	B6:BOOL;
	B7:BOOL;
END_VAR
VAR
	Bx : BYTE;
END_VAR

(*
version 1.0	4 aug 2006
programmer 	hugo
tested by		tobias

this function creates a byte from 8 individual bits

executioin TIME on wago 750-841 = 8 us
*)
BX.0 := B0;
BX.1 := B1;
BX.2 := B2;
BX.3 := B3;
BX.4 := B4;
BX.5 := B5;
BX.6 := B6;
BX.7 := B7;

Byte_of_bit := BX;
END_FUNCTION

(* POU Logic/gate logic/Byte_of_Dword, ST *)
FUNCTION Byte_of_Dword : BYTE
VAR_INPUT
	in : DWORD;
	N : BYTE;
END_VAR
VAR
	temp: DWORD;
END_VAR

(*
version 1.0	17 jan 2007
programmer 	hugo
tested by		tobias

this function extracts a single byte from the nth position from right (right is lowest byte) 
the lower byte (starting with Bit0 from in) is selected with N=0.
*)
temp := SHR(in,n*8);
Byte_of_Dword := DWORD_TO_BYTE(temp);
END_FUNCTION

(* POU Logic/gate logic/Byte_to_Bit, ST *)
FUNCTION_BLOCK Byte_to_Bit
VAR_INPUT
	IN: BYTE;
END_VAR
VAR_OUTPUT
	B0: BOOL;
	B1: BOOL;
	B2: BOOL;
	B3: BOOL;
	B4: BOOL;
	B5: BOOL;
	B6: BOOL;
	B7: BOOL;
END_VAR
VAR
END_VAR

(*
version 1.0	4 aug 2006
programmer 	hugo
tested by		tobias

this Function Block extracts the 8 Bits from a byte

executioin TIME on wago 750-841 = 13us
*)
B0 := IN.0;
B1 := IN.1;
B2 := IN.2;
B3 := IN.3;
B4 := IN.4;
B5 := IN.5;
B6 := IN.6;
B7 := IN.7;
END_FUNCTION_BLOCK

(* POU Logic/gate logic/check_parity, ST *)
FUNCTION check_parity : BOOL
VAR_INPUT
	in : DWORD;
	p : BOOL;
END_VAR
VAR
	cnt: INT := 0;
END_VAR

(*
version 1.1	10 sep 2007
programmer 	hugo
tested by		tobias

this function checks for an even partity for a dword and partity bit.

*)
WHILE in > 0 DO
	IF in.0 THEN cnt := cnt + 1; END_IF;
	in := SHR(in,1);
END_WHILE;
check_parity := even(cnt) XOR P;

(* revision history

rev 1.0 HM  1.oct.2006

rev 1.1 hm	10.sep.2007
	changed algorithm to improove performance

*)
END_FUNCTION

(* POU Logic/gate logic/DEC_2, ST *)
FUNCTION_BLOCK DEC_2
VAR_INPUT
	D: BOOL;
	A: BOOL;
END_VAR
VAR_OUTPUT
	Q0: BOOL;
	Q1: BOOL;
END_VAR
VAR
END_VAR

(*
version 1.1	3 Mar 2007
programmer 	hugo
tested by		tobias

a bit input will be decoded to the two outputs Q0 or Q1
dependent on the value of A
A=0 decodes to Q0 and A=1 decodes to Q1

*)
Q0 := D AND NOT A;
Q1 := D AND A;

(* revision history
hm 3.3.2007	rev 1.1
	rewritten in ST for better compatibility

*)
END_FUNCTION_BLOCK

(* POU Logic/gate logic/DEC_4, ST *)
FUNCTION_BLOCK DEC_4
VAR_INPUT
	D: BOOL;
	A0: BOOL;
	A1: BOOL;
END_VAR
VAR_OUTPUT
	Q0: BOOL;
	Q1: BOOL;
	Q2: BOOL;
	Q3: BOOL;
END_VAR
VAR
END_VAR

(*
version 1.1	3 Mar 2007
programmer 	hugo
tested by		tobias

a bit input will be decoded to one of the 4 outputs
dependent on the Adress on A0 and A1

executioin TIME on wago 750-841 = 9us
*)
Q0 := D AND NOT A0 AND NOT A1;
Q1 := D AND A0 AND NOT A1;
Q2 := D AND NOT A0 AND A1;
Q3 := D AND A0 AND A1;

(* revision history
hm 3.3.2007	rev 1.1
	rewritten in ST for better compatibility

*)
END_FUNCTION_BLOCK

(* POU Logic/gate logic/DEC_8, ST *)
FUNCTION_BLOCK DEC_8
VAR_INPUT
	D: BOOL;
	A0: BOOL;
	A1: BOOL;
	A2: BOOL;
END_VAR
VAR_OUTPUT
	Q0: BOOL;
	Q1: BOOL;
	Q2: BOOL;
	Q3: BOOL;
	Q4: BOOL;
	Q5: BOOL;
	Q6: BOOL;
	Q7: BOOL;
END_VAR
VAR
END_VAR

(*
version 1.1	3 mar 2007
programmer 	hugo
tested by		tobias

a bit input will be decoded to one of the 8 outputs
dependent on the Adress on A0, A1 and A2

executioin TIME on wago 750-841 = 17us
*)
Q0 := D AND NOT A0 AND NOT A1 AND NOT A2;
Q1 := D AND A0 AND NOT A1 AND NOT A2;
Q2 := D AND NOT A0 AND A1 AND NOT A2;
Q3 := D AND A0 AND A1 AND NOT A2;
Q4 := D AND NOT A0 AND NOT A1 AND A2;
Q5 := D AND A0 AND NOT A1 AND A2;
Q6 := D AND NOT A0 AND A1 AND A2;
Q7 := D AND A0 AND A1 AND A2;

(* revision history
hm 3.3.2007	rev 1.1
	rewritten in ST for better compatibility

*)
END_FUNCTION_BLOCK

(* POU Logic/gate logic/DWord_of_Byte, ST *)
FUNCTION DWord_of_Byte : DWORD
VAR_INPUT
	B0 : BYTE;
	B1 : BYTE;
	B2 : BYTE;
	B3 : BYTE;
END_VAR
VAR
END_VAR

(*
version 1.0	24 jan 2007
programmer 	hugo
tested by		tobias

this function creates a Dword from 4 individual bytes

*)
DWord_of_Byte := B3;
DWord_of_Byte := SHL(DWord_of_Byte,8) OR B2;
DWord_of_Byte := SHL(DWord_of_Byte,8) OR B1;
DWord_of_Byte := SHL(DWord_of_Byte,8) OR B0;
END_FUNCTION

(* POU Logic/gate logic/mux_2, ST *)
FUNCTION mux_2 : BOOL
VAR_INPUT
	D0: BOOL;
	D1: BOOL;
	A0: BOOL;
END_VAR
VAR
END_VAR

(*
	version 1.1	5 oct 2006
	programmer 	hugo
	tested BY		tobias

	dual input multiplexer
	depending on the value of A0, D0 or D1 will be switched to the Output

	executioin TIME on wago 750-841 = 7us
*)
mux_2 := (D0 AND NOT A0) OR (D1 AND A0);

(*

change history:
5.10.2006		rev 1.1
	changed to ST Langage for better protability.

*)
END_FUNCTION

(* POU Logic/gate logic/mux_4, ST *)
FUNCTION mux_4 : BOOL
VAR_INPUT
	D0: BOOL;
	D1: BOOL;
	D2: BOOL;
	D3: BOOL;
	A0: BOOL;
	A1: BOOL;
END_VAR
VAR
END_VAR

(*
	version 1.1	5 oct 2006
	programmer 	hugo
	tested BY		tobias

	quad input multiplexer
	depending on the value of A0 and A1, one of the 4 inputs will be switched to the Output

	executioin TIME on wago 750-841 = 13us
*)
mux_4 := (D0 AND NOT A0 AND NOT A1)
	OR (D1 AND A0 AND NOT A1)
	OR (D2 AND NOT A0 AND A1)
	OR (D3 AND A0 AND A1);


(* change history:

5.10.2006		rewritten to ST for better portability


*)
END_FUNCTION

(* POU Logic/gate logic/parity, ST *)
FUNCTION parity : BOOL
VAR_INPUT
	in : DWORD;
END_VAR
VAR
	cnt : INT := 0;
END_VAR

(*
	version 1.1	10 sep 2007
	programmer 	hugo
	tested BY		hans

this function calculates the even parity of an input Dword
the output will be true if the amount of high bits are an odd number.

*)
WHILE in > 0 DO
	IF in.0 THEN cnt := cnt +1; END_IF;
	in := SHR(in,1);
END_WHILE;
IF (cnt MOD 2) = 1 THEN parity := TRUE; ELSE parity := FALSE; END_IF;

(* revision history

rev 1.0 hm 1 sep 2006
	original version

rev 1.1 hm 10.9.2007
	changed algorithm to improove performance

*)
END_FUNCTION

(* POU Logic/gate logic/reverse, ST *)
FUNCTION reverse : BYTE
VAR_INPUT
	IN : BYTE;
END_VAR
VAR
END_VAR

(*
	version 1.0	9. oct 2006
	programmer 	hugo
	tested BY		tobias

This function reverses the bits of a byte so that afdter execution bit 7 is at bit 0 location and so forth.

*)
reverse.7 := in.0;
reverse.6 := in.1;
reverse.5 := in.2;
reverse.4 := in.3;
reverse.3 := in.4;
reverse.2 := in.5;
reverse.1 := in.6;
reverse.0 := in.7;


(* revision history
hm		9.oct 2007	rev 1.0
	original version

*)
END_FUNCTION

(* POU Logic/gate logic/SHL1, ST *)
FUNCTION SHL1 : DWORD
VAR_INPUT
	IN : DWORD;
	N : INT;
END_VAR
VAR CONSTANT
	temp : DWORD := 1;
END_VAR

(*
version 1.0	14 sep 2007
programmer 	hugo
tested by		tobias

SHL1 shifts N bits to the left filling the new bits with 1

*)
IF N = 32 THEN
	SHL1 := 16#FF_FF_FF_FF;
ELSE
	SHL1 := SHL(IN,N) OR SHL(temp,N)-1;
END_IF;

(* revision history
hm	14.9.2007	rev 1.0
	original version

*)
END_FUNCTION

(* POU Logic/gate logic/SHR1, ST *)
FUNCTION SHR1 : DWORD
VAR_INPUT
	IN : DWORD;
	N : INT;
END_VAR
VAR CONSTANT
	temp : DWORD := 2#11111111_11111111_11111111_11111111;
END_VAR

(*
version 1.0	14 sep 2007
programmer 	hugo
tested by		tobias

SHR1 shifts N bits to the right filling the new bits with 1

*)
IF N = 0 THEN
	SHR1 := in;
ELSE
	SHR1 := SHR(IN,N) OR SHL(temp,32-N);
END_IF;

(* revision history
hm	14.9.2007	rev 1.0
	original version

*)
END_FUNCTION

(* POU Logic/gate logic/Word_of_Byte, ST *)
FUNCTION Word_of_Byte : WORD
VAR_INPUT
	B0 : BYTE;
	B1 : BYTE;
END_VAR
VAR
END_VAR

(*
version 1.0	24 jan 2007
programmer 	hugo
tested by		tobias

this function creates a word from 2 individual bytes

*)
Word_of_Byte := B1;
Word_of_Byte := SHL(Word_of_Byte,8) + B0;
END_FUNCTION

(* POU Logic/gate logic/Word_of_Dword, ST *)
FUNCTION Word_of_Dword : WORD
VAR_INPUT
	in : DWORD;
	N : BYTE;
END_VAR
VAR
	temp: DWORD;
END_VAR

(*
version 1.0	17 jan 2007
programmer 	hugo
tested by		tobias

this function extracts a single word from the nth position from right (right is lowest byte)
the lower word (starting weith Bit0 from in) is selected with N=0.
*)
temp := SHR(in,n*16);
Word_of_Dword := DWORD_TO_WORD(temp);
END_FUNCTION

(* POU Logic/generators/B_TRIG, ST *)
FUNCTION_BLOCK B_TRIG
VAR_INPUT
	CLK : BOOL;
END_VAR
VAR_OUTPUT
	Q : BOOL := 0;
END_VAR
VAR
	edge : BOOL := 0;
END_VAR

(*
version 1.0	4 aug 2006
programmer 	hugo
tested by		tobias

this block is similar to R_trig and F_trig but it generates a pulse on rising and falling edge.

executioin TIME on wago 750-841 = 5us
*)
Q := clk XOR edge;
edge := CLK;
END_FUNCTION_BLOCK

(* POU Logic/generators/CLK_1ms, ST *)
FUNCTION_BLOCK CLK_1ms
VAR_INPUT
END_VAR
VAR_OUTPUT
	Q : BOOL;
END_VAR
VAR
	CLK : BOOL;
	edge : BOOL := 0;
	stime: DWORD;
END_VAR

(*
version 1.1	17 sep 2007
programmer 	hugo
tested by		tobias

clk_gen uses the internal sps time to generate one pulse every 1 ms
every pulse is only valid for one cycle so that a edge trigger is not necessary
clk_gen generates pulses depending on the accuracy of the system clock.

be careful, 1ms clocks will only work on very powerful sps cpu's
wago 750 - 841 will work with pulse width >= 10ms
*)
stime := T_PLC_MS();
clk := stime.0;
Q := clk XOR edge;
edge := CLK;

(* revision history
hm	4. aug 2006		rev 1.0
	original version

hm	17. sep 2007	rev 1.1
	replaced time() with T_PLC_MS() for compatibility reasons

*)
END_FUNCTION_BLOCK

(* POU Logic/generators/CLK_2ms, ST *)
FUNCTION_BLOCK CLK_2ms
VAR_INPUT
END_VAR
VAR_OUTPUT
	Q : BOOL;
END_VAR
VAR
	CLK : BOOL;
	edge : BOOL := 0;
	stime: DWORD;
END_VAR

(*
version 1.1	17 sep 2007
programmer 	hugo
tested by		tobias

clk_gen uses the internal sps time to generate one pulse every 2 ms
every pulse is only valid for one cycle so that a edge trigger is not necessary
clk_gen generates pulses depending on the accuracy of the system clock.

be careful, 1ms clocks will only work on very powerful sps cpu's
wago 750 - 841 will work with pulse width >= 10ms
*)
stime := T_PLC_MS();
clk := stime.1;
Q := clk XOR edge;
edge := CLK;

(* revision history
hm	4. aug 2006		rev 1.0
	original version

hm	17. sep 2007	rev 1.1
	replaced time() with T_PLC_MS() for compatibility reasons

*)
END_FUNCTION_BLOCK

(* POU Logic/generators/CLK_4ms, ST *)
FUNCTION_BLOCK CLK_4ms
VAR_INPUT
END_VAR
VAR_OUTPUT
	Q : BOOL;
END_VAR
VAR
	CLK : BOOL;
	edge : BOOL := 0;
	stime: DWORD;
END_VAR

(*
version 1.1	17 sep 2007
programmer 	hugo
tested by		tobias

clk_gen uses the internal sps time to generate one pulse every 4 ms
every pulse is only valid for one cycle so that a edge trigger is not necessary
clk_gen generates pulses depending on the accuracy of the system clock.

be careful, 1ms clocks will only work on very powerful sps cpu's
wago 750 - 841 will work with pulse width >= 10ms
*)
stime := T_PLC_MS();
clk := stime.2;
Q := clk XOR edge;
edge := CLK;

(* revision history
hm	4. aug 2006		rev 1.0
	original version

hm	17. sep 2007	rev 1.1
	replaced time() with T_PLC_MS() for compatibility reasons

*)
END_FUNCTION_BLOCK

(* POU Logic/generators/CLK_8ms, ST *)
FUNCTION_BLOCK CLK_8ms
VAR_INPUT
END_VAR
VAR_OUTPUT
	Q : BOOL;
END_VAR
VAR
	CLK : BOOL;
	edge : BOOL := 0;
	stime: DWORD;
END_VAR

(*
version 1.1	17 sep 2007
programmer 	hugo
tested by		tobias

clk_gen uses the internal sps time to generate one pulse every 8 ms
every pulse is only valid for one cycle so that a edge trigger is not necessary
clk_gen generates pulses depending on the accuracy of the system clock.

be careful, 1ms clocks will only work on very powerful sps cpu's
wago 750 - 841 will work with pulse width >= 10ms
*)
stime := T_PLC_MS();
clk := stime.3;
Q := clk XOR edge;
edge := CLK;

(* revision history
hm	4. aug 2006		rev 1.0
	original version

hm	17. sep 2007	rev 1.1
	replaced time() with T_PLC_MS() for compatibility reasons

*)
END_FUNCTION_BLOCK

(* POU Logic/generators/clk_div, ST *)
FUNCTION_BLOCK clk_div
VAR_INPUT
	clk : BOOL;
	rst: BOOL;
END_VAR
VAR_OUTPUT
	Q0 : BOOL := 0;
	Q1 : BOOL := 0;
	Q2 : BOOL := 0;
	Q3 : BOOL := 0;
	Q4 : BOOL := 0;
	Q5 : BOOL := 0;
	Q6 : BOOL := 0;
	Q7 : BOOL := 0;
END_VAR
VAR
	cnt: BYTE := 0;
END_VAR

(*
version 1.0	4 aug 2006
programmer 	hugo
tested by		tobias

this is a clock divider
each output divides the signal by 2
Q0 = clk / 2 , Q1 = Q0 / 2 and so on.
the outputs have a 50% duty cycle each.


*)
IF clk AND NOT rst THEN
	cnt:= cnt +1;
	Q0 := cnt.0;
	Q1 := cnt.1;
	Q2 := cnt.2;
	Q3 := cnt.3;
	Q4 := cnt.4;
	Q5 := cnt.5;
	Q6 := cnt.6;
	Q7 := cnt.7;
END_IF;
IF rst THEN
	cnt:= 0;
	Q0 := 0;
	Q1 := 0;
	Q2 := 0;
	Q3 := 0;
	Q4 := 0;
	Q5 := 0;
	Q6 := 0;
	Q7 := 0;
END_IF;
END_FUNCTION_BLOCK

(* POU Logic/generators/CLK_Pulse, ST *)
FUNCTION_BLOCK CLK_Pulse
VAR_INPUT
	PT : TIME := t#10ms;
	N : INT := 0;
	rst : BOOL := 0;
END_VAR
VAR_OUTPUT
	Q : BOOL := 0;
	cnt : INT := 0;
	run : BOOL := 0;
END_VAR
VAR
	pti : TIME := t#0ms;
	next_pulse: TIME := T#0s;
	overflow: BOOL := FALSE;
	tx: TIME;
END_VAR

(*
version 1.1	17 sep 2007
programmer 	hugo
tested by		tobias

clk_pulse uses the internal sps time to generate a clock with programmable period time.
the period time is defined for 10ms .. 65s.
pulse generation is continuous if N = 0 and for n pulses otherwise.
if the period time is set to less then 10ms the min clock perid is 10ms.
the first cycle after start is a clk pulse and then depending on the programmed period time a delay.
every pulse is only valid for one cycle so that a edge trigger is not necessary
clk_prg depending on the accuracy of the system clock.

*)
(* read system *)
tx := DWORD_TO_TIME(T_PLC_MS());


IF rst THEN
	run := FALSE;
	pti := t#0ms;
	next_pulse := t#0ms;
	overflow := FALSE;
	Q := FALSE;
	cnt := 0;
ELSIF cnt <= N OR N = 0 THEN
	IF NOT run THEN
		next_pulse := tx;
		run := TRUE;
		IF pt < T#10ms THEN PTI := T#10ms; ELSE pti := pt; END_IF;
	END_IF;
	IF tx >= next_pulse AND NOT overflow AND (cnt < N OR N = 0) THEN
		Q := TRUE;
		cnt := cnt + 1;
		IF next_pulse + pti < next_pulse THEN
			overflow := TRUE;
		END_IF;
		next_pulse := next_pulse + pti;
	ELSE
		Q := FALSE;
		IF cnt = N THEN run := FALSE; END_IF
		IF tx <= next_pulse THEN overflow := FALSE; END_IF;
	END_IF;
END_IF

(* revision history
hm		4. aug 2006		rev 1.0
	original version

hm		17. sep 2007	rev 1.1
	replaced time() with T_PLC_S() fr compatblity reasons

*)
END_FUNCTION_BLOCK

(* POU Logic/generators/D_Trig, ST *)
FUNCTION_BLOCK D_Trig
VAR_INPUT
	in : DWORD;
END_VAR
VAR_OUTPUT
	Q : BOOL;
	X : DWORD;
END_VAR
VAR
	last_in : DWORD;
END_VAR

(*
version 1.0	4 Sep 2007
programmer 	hugo
tested by		tobias

this block is similar to the IEC Standard R_trig and F_trig but it monitors a DWORD, WORD or Byte Variable instead and generated an Output Pulse for one cycle only when the input has changed.
an additional output x (Dword) will state the chage of the input.
Example: the input has chaged from 0001 to 0010 then the output x will be 2.

*)
IF (in XOR last_in) <> 0 THEN
	Q := TRUE;
	X := in - last_in;
	last_in := in;
ELSE
	Q := FALSE;
END_IF;


(* revision history

hm 4.09.2007	rev 1.0
	original version released

*)
END_FUNCTION_BLOCK

(* POU Logic/generators/gen_bit, ST *)
FUNCTION_BLOCK gen_bit
VAR_INPUT
	in0 : DWORD;
	in1 : DWORD;
	in2 : DWORD;
	in3 : DWORD;
	clk : BOOL := 0;
	steps : INT;
	rep : INT := 0;
	rst : BOOL := 0;
END_VAR
VAR_OUTPUT
	Q0 :BOOL := 0;
	Q1 :BOOL := 0;
	Q2 :BOOL := 0;
	Q3 :BOOL := 0;
	cnt : INT := 0;
	run : BOOL := 0;
END_VAR
VAR
	r0: DWORD;
	r1: DWORD;
	r2: DWORD;
	r3: DWORD;
	rx : INT := 1;
END_VAR

(*
version 1.0	4 aug 2006
programmer 	hugo
tested by		tobias

gen_bit is 4 bit sequencial pattern generator with 4 DWORD inputs and 4 serial outputs.
with the first clock pulse after a reset or after power on, bit 0 of the input DWORDS IN is present on the Outputs Q and the next clock cycle shifts to Bit 1 and so on.
the input steps defines how many bits of the input dwords will be shifted to the outputs. the sequence can be repetive when rep = 0 or any amount of repetitions can be defined with input rep.

*)
(* check if number of runs is finished or rep = 0 which means continuous *)

IF clk AND NOT rst THEN
	IF (rep = 0) OR (rx <= rep) THEN run := TRUE; ELSE run := FALSE; END_IF;
	IF run THEN
		(* check for step counter reached and reset to 0 if cnt = steps *)
		IF cnt = steps THEN
			cnt := 0;
		END_IF;

		(* when cnt = 0 then reload the inputs into the registers *)
		IF cnt = 0 THEN
			r0 := in0;
			r1 := in1;
			r2 := in2;
			r3 := in3;
		END_IF;

		(* when cnt < steps, shift the lowest bits to the outputs *)
		IF (cnt < steps) THEN
			Q0 := r0.0;
			Q1 := r1.0;
			Q2 := r2.0;
			Q3 := r3.0;
			r0 := SHR(r0,1);
			r1 := SHR(r1,1);
			r2 := SHR(r2,1);
			r3 := SHR(r3,1);
		END_IF;

		(* increment the step counter *)
		cnt := cnt +1;
		IF (cnt = steps) AND (rep <> 0) THEN rx := rx +1; END_IF;
		IF (rx > rep) AND (rep <> 0) THEN run := FALSE; END_IF;
	END_IF;
ELSE
	IF rst THEN
		Q0 := FALSE;
		Q1 := FALSE;
		Q2 := FALSE;
		Q3 := FALSE;
		r0 := 0;
		r1 := 0;
		r2 := 0;
		r3 := 0;
		cnt := 0;
		run := FALSE;
		rx := 1;
	END_IF;
END_IF;
END_FUNCTION_BLOCK

(* POU Logic/generators/gen_SQ, ST *)
FUNCTION_BLOCK gen_SQ
VAR_INPUT
	PT : TIME := T#0ms;
END_VAR
VAR_OUTPUT
	Q : BOOL := 0;
END_VAR
VAR
	pti : TIME := t#0ms;
	run: BOOL := FALSE;
	next_edge: TIME := t#0ms;
	overflow: BOOL := 0;
	tx: TIME;
END_VAR

(*
version 1.1	17 sep 2007
programmer 	hugo
tested by		tobias

gen_sq generates square wave signal with programmable period time.
the period time is defined for 10ms .. 65s
if the period time is set to less then 10ms the min perid is 10ms.

*)
(* read system time *)
tx := DWORD_TO_TIME(T_PLC_MS());

IF NOT run THEN
	next_edge := Tx;
	run := TRUE;
	IF pt < T#10ms THEN PTI := T#5ms; ELSE pti := pt / 2; END_IF;
END_IF;
IF (Tx >= next_edge) AND NOT overflow THEN
	Q := NOT Q;
	IF next_edge + pti < next_edge THEN
		(* time() will overflow every 50 days *)
		overflow := TRUE;
	END_IF;
	next_edge := next_edge + pti;
ELSE
	(* wait till time() has an overflow and reset overflow *)
	IF Tx <= next_edge THEN overflow := FALSE; END_IF;
END_IF;

(* revision history
hm	4. aug 2006		rev 1.0
	original version

hm	17. sep 2007	rev 1.1
	replaced time() with T_PLC_MS() for compatibility reasons

*)
END_FUNCTION_BLOCK

(* POU Logic/generators/sequence_4, ST *)
FUNCTION_BLOCK sequence_4
VAR_INPUT
	in0 : BOOL := TRUE;
	in1 : BOOL := TRUE;
	in2 : BOOL := TRUE;
	in3 : BOOL := TRUE;
	start : BOOL;
	rst : BOOL;
	wait0 : TIME := t#0s;
	delay0 : TIME := t#0s;
	wait1 : TIME := t#0s;
	delay1 : TIME := t#0s;
	wait2 : TIME := t#0s;
	delay2 : TIME := t#0s;
	wait3 : TIME := t#0s;
	delay3 : TIME := t#0s;
END_VAR
VAR_INPUT CONSTANT
	stop_on_error : BOOL := FALSE;
END_VAR
VAR_OUTPUT
	Q0 : BOOL;
	Q1 : BOOL;
	Q2 : BOOL;
	Q3 : BOOL;
	any : BOOL;
	run: BOOL;
	step : INT := -1;
	status : BYTE := 0;
END_VAR
VAR
	last : TIME;
	edge : BOOL;
	tx: TIME;
	init: BOOL;
END_VAR

(*
version 1.4	17 sep 2007
programmer 	oscat
tested by	hans

sequence_4 enables run when a low to high transition is present on start.
a low to high transition on start will restart the sequencer at any time while a rst will hold the sequencer in reset while true.
after run is enabled with a rising edge on start the sequencer waits for wait0 on in0 to enable q0 which stays on for delay0.
the next cycle starts with wait1, continues with delay 1 and so on...
if an edge is not detected during the wait period, the sequencer will then display the error number on the status output.
the status numbers 1..4 are errors in step 0..3.
after the last step that sets q3, the sequencer leaves q3 on for delay3 and then resets to the initial state.
a step output will indicate the current step of the sequencer and will also be present with a fault condition.
after the first output is turened on the sequencer switches from q0 to q1 and so on, at any time there is only one output enabled.
if an input signal is not detected during a wait period, the sequencer will display the error number ( 1 for in0, 2 for in1 .... ).
when an error is present and the config variable stop_on_error is set then the sequencer will stop. otherwise it will continue.
The status output will also display 110 for waiting and 111 for sequence running.
*)
(* read sps timer *)
tx := DWORD_TO_TIME(T_PLC_MS());

(* initialize on startup *)
IF NOT init THEN
	last := tx;
	init := TRUE;
	status := 110;
END_IF;

(* asynchronous reset *)
IF rst THEN
	step := -1;
	Q0 := 0;
	Q1 := 0;
	Q2 := 0;
	Q3 := 0;
	status := 110;
	run := 0;

(* edge on start input restarts the sequencer *)
ELSIF start AND NOT edge THEN
	step := 0;
	last := tx;
	status := 111;
	Q0 := 0;
	Q1 := 0;
	Q2 := 0;
	Q3 := 0;
	run := 1;
END_IF;
edge := start;

(* check if stop on status is necessary *)
IF status > 0 AND status < 100 AND stop_on_error THEN RETURN; END_IF;

(* sequence is running *)
IF run AND step = 0 THEN
	IF NOT q0 AND in0 AND tx - last <= wait0 THEN
		Q0 := TRUE;
		last := tx;
	ELSIF NOT q0 AND tx - last > wait0 THEN
		status := 1;
		run := FALSE;
	ELSIF q0 AND tx - last >= delay0 THEN
		step := 1;
		last := tx;
	END_IF;
END_IF;
IF run AND step = 1 THEN
	IF NOT q1 AND in1 AND tx - last <= wait1 THEN
		Q0 := FALSE;
		Q1 := TRUE;
		last := tx;
	ELSIF NOT q1 AND Tx - last > wait1 THEN
		status := 2;
		q0 := FALSE;
		run := FALSE;
	ELSIF q1 AND tx - last >= delay1 THEN
		step := 2;
		last := tx;
	END_IF;
END_IF;
IF run AND step = 2 THEN
	IF NOT q2 AND in2 AND tx - last <= wait2 THEN
		Q1 := FALSE;
		Q2 := TRUE;
		last := tx;
	ELSIF NOT q2 AND Tx - last > wait2 THEN
		status := 3;
		q1 := FALSE;
		run := FALSE;
	ELSIF q2 AND tx - last >= delay2 THEN
		step := 3;
		last := tx;
	END_IF;
END_IF;
IF run AND step = 3 THEN
	IF NOT q3 AND in3 AND tx - last <= wait3 THEN
		Q2 := FALSE;
		Q3 := TRUE;
		last := tx;
	ELSIF NOT q3 AND Tx - last > wait3 THEN
		status := 4;
		q2 := FALSE;
		run := FALSE;
	ELSIF q3 AND tx - last >= delay3 THEN
		step := -1;
		q3 := FALSE;
		run := FALSE;
		status := 110;
	END_IF;
END_IF;
any := q0 OR q1 OR q2 OR q3;

(*
hm 1.10.06		rev 1.1
	corrected delay logic to be after event and not before
	added any output

hm 1.12.06		rev 1.2
	corrected failure in sequence logic.
	added init at startup to prevent from initial error after start.

hm 17.1.2007		rev 1.3
	changed output fault to status for better compatibility with other modules (ESR).
	added stop on error functionality and setup variable
	default for inputs in0..3 is true.
	renamed variable state to step

hm	17.sep 2007		rev 1.4
	replaced time() with T_PLC_MS() for compatibility reasons

*)
END_FUNCTION_BLOCK

(* POU Logic/memory/FIFO_16, ST *)
FUNCTION_BLOCK FIFO_16
VAR_INPUT
	Din : DWORD;
	WR : BOOL;
	E : BOOL;
	RST : BOOL;
END_VAR
VAR_OUTPUT
	Dout : DWORD := 0;
	empty : BOOL := TRUE;
	full : BOOL := FALSE;
END_VAR
VAR
	fifo : ARRAY[0..15] OF DWORD;
	NW : INT := 0;
	NR : INT := 0;
	top : INT := 15;
END_VAR

(*
	version 1.0	4 aug 2006
	programmer 	hugo
	tested by		tobias

16 Dword FIFO memory
*)
IF rst THEN
	(* asynchronous reset for the fifo *)
	NW := 0;
	NR := 0;
	Dout := 0;
	empty := TRUE;
	full := FALSE;
ELSIF WR AND E AND NOT full THEN
	(* write action *)
	fifo[NW] := Din;
	IF NW = top THEN NW := 0; ELSE NW := NW + 1; END_IF
	IF NW = NR THEN full := TRUE; END_IF
	empty := FALSE;
ELSIF NOT WR AND E AND NOT empty THEN
	(* read from stack *)
	Dout := fifo[NR];
	IF NR = top THEN NR := 0; ELSE NR := NR + 1; END_IF;
	IF NR = NW THEN empty := TRUE; END_IF;
	full := FALSE;
END_IF;
END_FUNCTION_BLOCK

(* POU Logic/memory/FIFO_32, ST *)
FUNCTION_BLOCK FIFO_32
VAR_INPUT
	Din : DWORD;
	WR : BOOL;
	E : BOOL;
	RST : BOOL;
END_VAR
VAR_OUTPUT
	Dout : DWORD := 0;
	empty : BOOL := TRUE;
	full : BOOL := FALSE;
END_VAR
VAR
	fifo : ARRAY[0..31] OF DWORD;
	NW : INT := 0;
	NR : INT := 0;
	top : INT := 31;
END_VAR

(*
	version 1.0	4 aug 2006
	programmer 	hugo
	tested by		tobias

32 Dword FIFO memory
*)
IF rst THEN
	(* asynchronous reset for the fifo *)
	NW := 0;
	NR := 0;
	Dout := 0;
	empty := TRUE;
	full := FALSE;
ELSIF WR AND E AND NOT full THEN
	(* write action *)
	fifo[NW] := Din;
	IF NW = top THEN NW := 0; ELSE NW := NW + 1; END_IF
	IF NW = NR THEN full := TRUE; END_IF
	empty := FALSE;
ELSIF NOT WR AND E AND NOT empty THEN
	(* read from stack *)
	Dout := fifo[NR];
	IF NR = top THEN NR := 0; ELSE NR := NR + 1; END_IF;
	IF NR = NW THEN empty := TRUE; END_IF;
	full := FALSE;
END_IF;
END_FUNCTION_BLOCK

(* POU Logic/memory/STACK_16, ST *)
FUNCTION_BLOCK STACK_16
VAR_INPUT
	Din : DWORD;
	RW : BOOL;
	E : BOOL;
	RST : BOOL;
END_VAR
VAR_OUTPUT
	Dout : DWORD := 0;
	empty : BOOL := TRUE;
	full : BOOL := FALSE;
END_VAR
VAR
	Stack : ARRAY[0..15] OF DWORD;
	N : INT := -1;
	top : INT := 15;
END_VAR

(*
	version 1.0	4 aug 2006
	programmer 	hugo
	tested by		tobias

16 Dword STACK memory
*)
IF rst THEN
	(* asynchronous reset for the fifo *)
	N := -1;
	Dout := 0;
	empty := TRUE;
	full := FALSE;
ELSIF RW AND E AND NOT full THEN
	(* write action *)
	N := N + 1;
	IF N = top THEN full := TRUE; END_IF;
	empty := FALSE;
	stack[N] := Din;
ELSIF NOT RW AND E AND NOT empty THEN
	(* read from stack *)
	Dout := stack[N];
	N := N -1;
	IF N < 0 THEN empty := TRUE; END_IF;
	full := FALSE;
END_IF;
END_FUNCTION_BLOCK

(* POU Logic/memory/STACK_32, ST *)
FUNCTION_BLOCK STACK_32
VAR_INPUT
	Din : DWORD;
	RW : BOOL;
	E : BOOL;
	RST : BOOL;
END_VAR
VAR_OUTPUT
	Dout : DWORD := 0;
	empty : BOOL := TRUE;
	full : BOOL := FALSE;
END_VAR
VAR
	Stack : ARRAY[0..31] OF DWORD;
	N : INT := -1;
	top : INT := 31;
END_VAR

(*
	version 1.0	4 aug 2006
	programmer 	hugo
	tested by		tobias

32 Dword STACK memory
*)
IF rst THEN
	(* asynchronous reset for the fifo *)
	N := -1;
	Dout := 0;
	empty := TRUE;
	full := FALSE;
ELSIF RW AND E AND NOT full THEN
	(* write action *)
	N := N + 1;
	IF N = top THEN full := TRUE; END_IF;
	empty := FALSE;
	stack[N] := Din;
ELSIF NOT RW AND E AND NOT empty THEN
	(* read from stack *)
	Dout := stack[N];
	N := N -1;
	IF N < 0 THEN empty := TRUE; END_IF;
	full := FALSE;
END_IF;
END_FUNCTION_BLOCK

(* POU Logic/Others/CRC_CHECK, ST *)
FUNCTION CRC_CHECK : BOOL
VAR_INPUT
	pt : POINTER TO ARRAY[0..32000] OF BYTE;
	size : INT;
END_VAR
VAR_INPUT CONSTANT
	Polynom_L : DWORD;
	Polynom_32 : BOOL;
END_VAR
VAR
	temp: DWORD;
END_VAR

(*
version 1.0	9 jun 2007
programmer 	hugo
tested by		tobias

CRC_CHECK checks a block of data for a crc checksum and returns true is the checksum is 0 and therfore a error free data transmission.
the CRC Polynom is specified with the config variable Polynom_L which holds the lowest 32 bits of the polynom and Polynom_33 which holds bit 33 of the Polynom.
A Polynom x4 + X + 1 is represented by 10011.
The input data is an array of byte of any size, the function is called by CRC_CHECK(ADR(array),SIZEOF(array)).

*)
temp := CRC_GEN(pt, size, polynom_L, polynom_32, 0, 0, FALSE, FALSE);
IF temp = 0 THEN CRC_CHECK := TRUE; ELSE CRC_CHECK := FALSE; END_IF;

(* typical crc polynoms

CRC-4-ITU 			x4 + x + 1 					(ITU G.704, p. 12) 	0x3 or 0xC (0x9)
CRC-5-ITU 			x5 + x4 + x2 + 1 			(ITU G.704, p. 9) 	0x15 or 0x15 (0x0B)
CRC-5-USB 			x5 + x2 + 1 				(use: USB token packets) 	0x05 or 0x14 (0x9)
CRC-6-ITU 			x6 + x + 1 					(ITU G.704, p. 3) 	0x03 or 0x30 (0x21)
CRC-7 				x7 + x3 + 1 				(use: telecom systems, MMC) 	0x09 or 0x48 (0x11)
CRC-8-ATM 			x8 + x2 + x + 1 				(use: ATM HEC) 	0x07 or 0xE0 (0xC1)
CRC-8-CCITT 		x8 + x7 + x3 + x2 + 1 		(use: 1-Wire bus) 	0x8D or 0xB1 (0x63)
CRC-8-Dallas/Maxim 	x8 + x5 + x4 + 1 			(use: 1-Wire bus) 	0x31 or 0x8C (0x19)
CRC-8 				x8 + x7 + x6 + x4 + x2 + 1 	0xD5 or 0xAB (0x57)
CRC-8-SAE J1850 	x8 + x4 + x3 + x2 + 1 		0x1D or 0xB8
CRC-10 				x10 + x9 + x5 + x4 + x + 1 	0x233 or 0x331 (0x263)
CRC-12 				x12 + x11 + x3 + x2 + x + 1 (use: telecom systems) 	0x80F or 0xF01 (0xE03)
CRC-15-CAN 			x15 + x14 + x10 + x8 + x7 + x4 + x3 + 1 	0x4599 or 0x4CD1 (0x19A3)
CRC-16-Fletcher 	Not a CRC; see Fletcher's checksum 	Used in Adler-32 A & B CRCs
CRC-16-CCITT 	x16 + x12 + x5 + 1 (XMODEM,X.25, V.41, Bluetooth, PPP, IrDA; known as "CRC-CCITT") 	0x1021 or 0x8408 (0x0811)
CRC-16-IBM 	x16 + x15 + x2 + 1 (USB, many others; also known as "CRC-16") 	0x8005 or 0xA001 (0x4003)
CRC-24-Radix-64 	x24 + x23 + x18 + x17 + x14 + x11 + x10 + x7 + x6 + x5 + x4 + x3 + x + 1 	0x864CFB or 0xDF3261 (0xBE64C3)
CRC-32-Adler 	Not a CRC; see Adler-32 	See Adler-32
CRC-32-MPEG2 	x32 + x26 + x23 + x22 + x16 + x12 + x11 + x10 + x8 + x7 + x5 + x4 + x2 + x + 1 	0x04C11DB7 or 0xEDB88320 (0xDB710641) Also used in IEEE 802.3
CRC-32-IEEE 802.3 	x32 + x26 + x23 + x22 + x16 + x12 + x11 + x10 + x8 + x7 + x5 + x4 + x2 + x + 1 (V.42) 	0x04C11DB7 or 0xEDB88320 (0xDB710641)
CRC-32C (Castagnoli) 	x32 + x28 + x27 + x26 + x25 + x23 + x22 + x20 + x19 + x18 + x14 + x13 + x11 + x10 + x9 + x8 + x6 + 1 	0x1EDC6F41 or 0x82F63B78 (0x05EC76F1)
CRC-64-ISO 	x64 + x4 + x3 + x + 1 (use: ISO 3309) 	0x000000000000001B or 0xD800000000000000 (0xB000000000000001)
CRC-64-ECMA-182 	x64 + x62 + x57 + x55 + x54 + x53 + x52 + x47 + x46 + x45 + x40 + x39 + x38 + x37 + x35 + x33 + x32 + x31 + x29 + x27 + x24 + x23 + x22 + x21 + x19 + x17 + x13 + x12 + x10 + x9 + x7 + x4 + x + 1
(as described in ECMA-182 p.63) 	0x42F0E1EBA9EA3693 or 0xC96C5795D7870F42 (0x92D8AF2BAF0E1E85)

*)

(* revision history

hm		9.6.2007	rev 1.0		original version 

*)
END_FUNCTION

(* POU Logic/Others/CRC_GEN, ST *)
FUNCTION CRC_GEN : DWORD

VAR_INPUT
	pt : POINTER TO ARRAY[0..32000] OF BYTE;
	size : INT;
END_VAR
VAR_INPUT CONSTANT
	Polynom_L : DWORD;
	Polynom_32 : BOOL;
	init: DWORD := 0;
	XOR_out : DWORD;
	rev_in : BOOL;
	rev_out : BOOL;
END_VAR
VAR
	polynom : DWORD;
	p_length : INT;
	BS : BYTE;
	data : DWORD;
	count : BYTE;
	temp : BOOL;
	step: INT;
END_VAR

(*
version 1.2	9 oct 2007
programmer 	hugo
tested by		tobias

CRC_GEN generates a CRC checksum from a block of data and returns  the checksum in a DWORD to be connected to the data for transmission.
the CRC Polynom is specified with the config variable Polynom_L which holds the lowest 32 bits of the polynom and Polynom_33 which holds bit 33 of the Polynom.
A Polynom x4 + X + 1 is represented by 10011.
The input data is an array of byte of any size, the function is called by CRC_GEN(ADR(array),SIZEOF(array)).

*)
(* check for polynom length and calculate p_length polynom will be aligned to high side of word*)
polynom := polynom_L;
IF polynom_32 = 1 THEN
	p_length := 33;
ELSE;
	p_length := 32;
	WHILE Polynom.31 = 0 AND p_length > 0 DO
		p_length := p_length - 1;
		Polynom := SHL(polynom,1);
	END_WHILE;
	Polynom := SHL(polynom,1);
END_IF;


(* load start code and first data byte for crc calculation *)
data := init;
BS := pt^[0];
IF rev_in THEN bs := reverse(bs); END_IF;

(* calcualte checksum *)
WHILE step < size + 4 DO
	temp := data.31;
	data := SHL(data,1);
	data.0 := BS.7;
	bs := SHL(bs,1);
	count := count + 1;
	IF count = 8 THEN
		step := step + 1;
		count := 0;
		IF step < size THEN
			bs := pt^[step];
			IF rev_in THEN bs := reverse(bs); END_IF;
		END_IF;
	END_IF;
	(* check highest bit if true then xor polynom *)
	IF temp THEN data := data XOR polynom; END_IF;
END_WHILE;

(* reverse crc if necessary *)

IF rev_out THEN
	CRC_GEN.31 := data.31;
	FOR step := p_length TO 3 BY -1 DO
		data := SHL(data,1);
		CRC_GEN := SHR(CRC_GEN,1);
		CRC_GEN.31 := data.31;
	END_FOR;
ELSE
	CRC_GEN := data;
END_IF;

(* final XOR and align crc checksum to right side of dword *)
CRC_GEN := CRC_GEN XOR SHL(xor_out, 32 - p_length + 1);
CRC_GEN := SHR(CRC_GEN,32 - p_length + 1);



(* old code prior to rev 1.2
B1 := pt^[0];
IF size > 1 THEN B2 := pt^[1]; ELSE B2 := 0; END_IF;
IF size > 2 THEN B3 := pt^[2]; ELSE B3 := 0; END_IF;
IF size > 3 THEN B4 := pt^[3]; ELSE B4 := 0; END_IF;
IF size > 4 THEN BS := pt^[4]; ELSE BS := 0; END_IF;
data := DWord_of_Byte(B4,B3,B2,B1);

WHILE step < size DO
	temp := data.31;
	data := SHL(data,1);
	data.0 := BS.7;
	bs := SHL(bs,1);
	count := count + 1;
	IF count = 8 THEN
		step := step + 1;
		count := 0;
		IF step + 4 < size THEN bs := pt^[step+ 4]; END_IF;
	END_IF;
	(* check highest bit if true then xor polynom *)
	IF temp = TRUE THEN
		data := data XOR polynom;
	END_IF;
END_WHILE;

(* align crc checksum to right side of dword *)
CRC_GEN := SHR(data,32 - p_length +1);
*)


(* typical crc polynoms

CRC-4-ITU 			x4 + x + 1 					(ITU G.704, p. 12) 	0x3 or 0xC (0x9)
CRC-5-ITU 			x5 + x4 + x2 + 1 			(ITU G.704, p. 9) 	0x15 or 0x15 (0x0B) Bluetooth
CRC-5-USB 			x5 + x2 + 1 				(use: USB token packets) 	0x05 or 0x14 (0x9)
CRC-6-ITU 			x6 + x + 1 					(ITU G.704, p. 3) 	0x03 or 0x30 (0x21)
CRC-7 				x7 + x3 + 1 				(use: telecom systems, MMC) 	0x09 or 0x48 (0x11)
CRC-8-ATM 			x8 + x2 + x + 1 				(use: ATM HEC) 	0x07 or 0xE0 (0xC1)
CRC-8-CCITT 		x8 + x7 + x3 + x2 + 1 		(use: 1-Wire bus) 	0x8D or 0xB1 (0x63)
CRC-8-Dallas/Maxim 	x8 + x5 + x4 + 1 			(use: 1-Wire bus) 	0x31 or 0x8C (0x19)
CRC-8 				x8 + x7 + x6 + x4 + x2 + 1 	0xD5 or 0xAB (0x57)
CRC-8-SAE J1850 	x8 + x4 + x3 + x2 + 1 		0x1D or 0xB8
CRC-10 				x10 + x9 + x5 + x4 + x + 1 	0x233 or 0x331 (0x263)
CRC-12 				x12 + x11 + x3 + x2 + x + 1 (use: telecom systems) 	0x80F or 0xF01 (0xE03)
CRC-15-CAN 			x15 + x14 + x10 + x8 + x7 + x4 + x3 + 1 	0x4599 or 0x4CD1 (0x19A3)
CRC-16-Fletcher 	Not a CRC; see Fletcher's checksum 	Used in Adler-32 A & B CRCs
CRC-16-CCITT 	x16 + x12 + x5 + 1 (XMODEM,X.25, V.41, Bluetooth, PPP, IrDA; known as "CRC-CCITT") 	0x1021 or 0x8408 (0x0811)
CRC-16-IBM 	x16 + x15 + x2 + 1 (USB, many others; also known as "CRC-16") 	0x8005 or 0xA001 (0x4003)
CRC-24-Radix-64 	x24 + x23 + x18 + x17 + x14 + x11 + x10 + x7 + x6 + x5 + x4 + x3 + x + 1 	0x864CFB or 0xDF3261 (0xBE64C3)
CRC-32-Adler 	Not a CRC; see Adler-32 	See Adler-32
CRC-32-MPEG2 	x32 + x26 + x23 + x22 + x16 + x12 + x11 + x10 + x8 + x7 + x5 + x4 + x2 + x + 1 	0x04C11DB7 or 0xEDB88320 (0xDB710641) Also used in IEEE 802.3
CRC-32-IEEE 802.3 	x32 + x26 + x23 + x22 + x16 + x12 + x11 + x10 + x8 + x7 + x5 + x4 + x2 + x + 1 (V.42) 	0x04C11DB7 or 0xEDB88320 (0xDB710641)
CRC-32C (Castagnoli) 	x32 + x28 + x27 + x26 + x25 + x23 + x22 + x20 + x19 + x18 + x14 + x13 + x11 + x10 + x9 + x8 + x6 + 1 	0x1EDC6F41 or 0x82F63B78 (0x05EC76F1)
CRC-64-ISO 	x64 + x4 + x3 + x + 1 (use: ISO 3309) 	0x000000000000001B or 0xD800000000000000 (0xB000000000000001)
CRC-64-ECMA-182 	x64 + x62 + x57 + x55 + x54 + x53 + x52 + x47 + x46 + x45 + x40 + x39 + x38 + x37 + x35 + x33 + x32 + x31 + x29 + x27 + x24 + x23 + x22 + x21 + x19 + x17 + x13 + x12 + x10 + x9 + x7 + x4 + x + 1
(as described in ECMA-182 p.63) 	0x42F0E1EBA9EA3693 or 0xC96C5795D7870F42 (0x92D8AF2BAF0E1E85)

*)

(* revision history

hm		9.6.2007	rev 1.0		
	original version 

hm		11.9.2007	rev 1.1
	deleted unused variable i



hm		9. oct 2007 rev 1.2
	added init code for crc and xor_out
	added refelct in and reflect_out (rev_in und Rev_out)

*)
END_FUNCTION

(* POU Logic/Others/matrix, ST *)
FUNCTION_BLOCK matrix
VAR_INPUT
	x1, x2, x3, x4, X5 : BOOL;
END_VAR
VAR_INPUT CONSTANT
	Release : BOOL;
END_VAR
VAR_OUTPUT
	code : BYTE;
	TP : BOOL;
	y1: BOOL := TRUE;
	y2, y3, y4 : BOOL;
END_VAR
VAR
	line : BYTE := 1;
	X : ARRAY[1..4] OF BYTE; (* scan line inputs *)
	L : ARRAY[1..4] OF BYTE; (* scan line status *)
	i: INT;
	temp: BYTE;
END_VAR

(*
version 1.1	11 sep 2007
programmer 	hugo
tested by		tobias

MATRIX is a matrix keyboard encoder for 4 rows and up to 5 columns.
matrix can send a code while a key is pressed and it sends another code while a key is released when the setup variable 'release' is set to true.
the setup variable release is false the code is only sent when the key is pressed.
the output byte holds the 5 columns in the lowest bits 0..2  and the row number in bits 4..6, while bit 7 is true for a key pressed and false for a key released.

*)
TP := FALSE;
code := 0;

(* read scan lines *)
X[line].0 := X1;
X[line].1 := X2;
X[line].2 := X3;
X[line].3 := X4;
X[line].4 := X5;

(* compare for change *)
FOR i := 1 TO 4 DO
	IF X[i] <> L[i] THEN
		(* scan line information has changed code need to be found and generated *)
		temp := x[i] XOR L[i];
		IF temp.0 THEN
			code := 1;
			code.7 := X[i].0;
			L[i].0 := X[i].0;
		ELSIF temp.1 THEN
			code := 2;
			code.7 := X[i].1;
			L[i].1 := X[i].1;
		ELSIF temp.2 THEN
			code := 3;
			code.7 := X[i].2;
			L[i].2 := X[i].2;
		ELSIF temp.3 THEN
			code := 4;
			code.7 := X[i].3;
			L[i].3 := X[i].3;
		ELSIF temp.4 THEN
			code := 5;
			code.7 := X[i].4;
			L[i].4 := X[i].4;
		END_IF;
		i := 5;
		TP := TRUE;
		Code.4 := Line.0;
		Code.5 := Line.1;
		Code.6 := Line.2;

		(* check if release codes need to be killed *)
		IF NOT release AND code < 127 THEN
			code := 0;
			TP := 0;
		END_IF;
	END_IF;
END_FOR;

(* increment scan line every cycle *)
CASE line OF
	1 :	Line := 2;
		Y1 := FALSE; Y3 := FALSE; Y4 := FALSE; Y2 := TRUE;
	2 :	Line := 3;
		Y1 := FALSE; Y2 := FALSE; Y4 := FALSE; Y3 := TRUE;
	3 :	Line := 4;
		Y1 := FALSE; Y2 := FALSE; Y3 := FALSE; Y4 := TRUE;
	4 :	Line := 1;
		Y2 := FALSE; Y3 := FALSE; Y4 := FALSE; Y1 := TRUE;
END_CASE;

(* revision history
hm		10.6.2007	rev 1.0		
	original version 


hm		11.9.2007	rev 1.1		
	deleted unused variables k and old_code
*)
END_FUNCTION_BLOCK

(* POU mathematical/array functions/_array_init, ST *)
FUNCTION _array_init : BOOL
VAR_INPUT
	pt : POINTER TO ARRAY[0..32000] OF REAL;
	size : INT;
	init : REAL;
END_VAR
VAR
	i: INT;
	stop: INT;
END_VAR


(*
version 1.2	14 nov 2007
programmer 	hugo
tested by		tobias

this function will initialize a given array with a value init.
the function needs to be called:	_array_init(adr("array"),sizeof("array"));
this function will manipulate a given array.
the function manipulates the original array, it rerturnes true when finished.
because this function works with pointers its very time efficient and it needs no extra memory.

*)
stop := SHR(size,2)-1;
FOR i := 0 TO stop DO
	pt^[i] := init;
END_FOR;
_array_init := TRUE;

(* revision History

hm 6.1.2007		rev 1.1
	change type of function to bool
	added  array_init := true to set output true.

hm	14.11.2007	rev 1.2
	changed stop calculation to be more efficient
*)
END_FUNCTION

(* POU mathematical/array functions/_array_median, ST *)
FUNCTION _array_median : REAL
VAR_INPUT
	pt : POINTER TO ARRAY[0..32000] OF REAL;
	size : INT;
END_VAR
VAR
	i: INT;
	stop: INT;
END_VAR

(*
version 1.4	14 nov 2007
programmer 	hugo
tested by		tobias

this function will calculate the median of a given array.
in order to do so the ariginal array is sorted and stays sorted after the function finishes
the function needs to be called:	_array_median(adr("array"),sizeof("array"));
this function will manipulate a given array.
the function will return the median of the original array.
for example [12,0,4,7,1] the median is 4 and the array after the function is called is [0,1,4,7,12]
because this function works with pointers its very time efficient and it needs no extra memory.

*)
_array_sort(pt,size);
stop := SHR(size,2)-1;
IF even(stop) THEN
	_array_median := pt^[stop/2];
ELSE
	i := SHR(stop,1);
	_array_median := (pt^[i] + pt^[i+1])/2;
END_IF;

(* old code
stop := (size - SIZEOF(pt)) / SIZEOF(pt);
FOR i := 0 TO stop - 1 DO
	FOR m := i + 1 TO stop DO
		IF pt^[i] > pt^[m] THEN
			temp := pt^[i];
			pt^[i] := pt^[m];
			pt^[m] := temp;
		END_IF;
	END_FOR;
END_FOR;
IF even(stop) THEN
	_array_median := pt^[stop/2];
ELSE
	i := stop/2;
	_array_median := (pt^[i] + pt^[i+1])/2;
END_IF;
*)
(* revision history
hm 	3.3.2007		rev 1.1
	corrected an error, changed the statement line 14	i := TRUNC(stop/2); to i := stop/2;

hm		22. sep 2007	rev 1.2
	changed algorithm to use _array_soft for performance reasons

hm		8. oct 2007		rev 1.3
	deleted unused variables m and temp

hm		14. nov 2007		rev 1.4
	corrected a problem with size calculation
*)
END_FUNCTION

(* POU mathematical/array functions/_array_sort, ST *)
FUNCTION _array_sort : BOOL
VAR_INPUT
	f : POINTER TO ARRAY[1..32000] OF REAL;
	size : INT;
END_VAR
VAR
	i: INT;
	j: INT;
	temp : REAL;
	stop : INT;
	heapsize: INT;
	popmax : REAL;
	size2: INT;
END_VAR

(*
version 1.3	14 nov 2007
programmer 	hugo
tested by		tobias

this function will sort a given array.
the function needs to be called:	_array_sort(adr("array"),sizeof("array"));
this function will manipulate a given array.
the function will not return anything except true, it will instead manipulate the original array.
because this function works with pointers its very time efficient and it needs no extra memory.

*)
(* generate heap *)

size := SHR(size,2);
size2 := SHR(size,1);
FOR i := SIZE2  TO 1 BY -1 DO 		(* zweite Hälfte des Feldes braucht nicht betrachtet werden *)
	j:=i;
    WHILE j <= SIZE2 DO
     	stop := j * 2 + 1;               (* finde Maximum der (beiden) Söhne *)
        IF stop > SIZE THEN stop := stop - 1;
        ELSIF f^[stop-1] > f^[stop] THEN stop := stop - 1;
		END_IF;
        IF f^[j] < f^[stop] THEN   		(* ggf. tauschen *)
         	temp := f^[j];
            f^[j] := f^[stop];
            f^[stop] := temp;
        END_IF;
        j := stop;
    END_WHILE;
END_FOR;

(* heapsort *)
FOR heapsize := size TO 1 BY -1 DO
	popmax := f^[1];
	f^[1] := f^[heapsize];
   	i := 1;
	WHILE i <= (heapsize / 2) DO	     (* letztes Element an Anfang setzen und versickern lassen *)
       	stop := i * 2 + 1;                (* finde Maximum der (beiden) Söhne *)
        	IF stop > heapsize THEN stop := stop - 1;
        	ELSIF f^[stop-1] > f^[stop] THEN stop := stop - 1;
	 	END_IF;
        	IF f^[i] < f^[stop] THEN	     (* ggf. tauschen *)
            		temp := f^[i];
            		f^[i] := f^[stop];
            		f^[stop] := temp;
        	END_IF;
        	i := stop;
    	END_WHILE;
	f^[heapsize] := popmax;
END_FOR;


(* old algorithm bubble sort used before rev 1.2
stop := (size - SIZEOF(pt)) / SIZEOF(pt);
FOR i := 0 TO stop - 1 DO
	FOR m := i + 1 TO stop DO
		IF pt^[i] > pt^[m] THEN
			temp := pt^[i];
			pt^[i] := pt^[m];
			pt^[m] := temp;
		END_IF;
	END_FOR;
END_FOR;
_array_sort := TRUE;

*)
(* revision history

hm 6.1.2007 	rev 1.1
	changed return value to true

hm	22. sep 2007	rev 1.2
	changed sorting algorithm to heap sort for performance reasons

hm 14. nov 2007	rev 1.3
	changed calculation of stop to be more efficient

*)
END_FUNCTION

(* POU mathematical/array functions/array_avg, ST *)
FUNCTION array_avg : REAL
VAR_INPUT
	pt : POINTER TO ARRAY[0..32000] OF REAL;
	size : INT;
END_VAR
VAR
	i: INT;
	stop: INT;
END_VAR

(*
version 1.0	2 oct 2006
programmer 	hugo
tested by		tobias

this function will calculate the average of a given array.
the function needs to be called:	array_avg(adr("array"),sizeof("array"));
because this function works with pointers its very time efficient and it needs no extra memory.

*)
stop := (size -SIZEOF(pt)) / SIZEOF(pt);
array_avg := pt^[0];
FOR i := 1 TO stop DO
	array_avg := array_avg + pt^[i];
END_FOR;
array_avg := array_avg / (stop + 1);
END_FUNCTION

(* POU mathematical/array functions/array_max, ST *)
FUNCTION array_max : REAL
VAR_INPUT
	pt : POINTER TO ARRAY[0..32000] OF REAL;
	size : INT;
END_VAR
VAR
	i: INT;
	stop: INT;
END_VAR

(*
version 1.0	2 oct 2006
programmer 	hugo
tested by		tobias

this function will calculate the max value of a given array.
the function needs to be called:	array_max(adr("array"),sizeof("array"));
because this function works with pointers its very time efficient and it needs no extra memory.

*)
stop := (size -SIZEOF(pt)) / SIZEOF(pt);
array_max := pt^[0];
FOR i := 1 TO stop DO
	IF pt^[i] > array_max THEN array_max := pt^[i]; END_IF;
END_FOR;
END_FUNCTION

(* POU mathematical/array functions/array_min, ST *)
FUNCTION array_min : REAL
VAR_INPUT
	pt : POINTER TO ARRAY[0..32000] OF REAL;
	size : INT;
END_VAR
VAR
	i: INT;
	stop: INT;
END_VAR

(*
version 1.0	2 oct 2006
programmer 	hugo
tested by		tobias

this function will calculate the min value of a given array.
the function needs to be called:	array_min(adr("array"),sizeof("array"));
because this function works with pointers its very time efficient and it needs no extra memory.

*)
stop := (size - SIZEOF(pt)) / SIZEOF(pt);
array_min := pt^[0];
FOR i := 1 TO stop DO
	IF pt^[i] < array_min THEN array_min := pt^[i]; END_IF;
END_FOR;
END_FUNCTION

(* POU mathematical/array functions/array_sdv, ST *)
FUNCTION array_sdv : REAL
VAR_INPUT
	pt : POINTER TO ARRAY[0..32000] OF REAL;
	size : INT;
END_VAR
VAR
END_VAR

(*
version 1.0	1 apr 2007
programmer 	hugo
tested by		tobias

this function will calculate the standard deviation of a given array.
the function needs to be called:	array_sdv(adr("array"),sizeof("array"));
because this function works with pointers its very time efficient and it needs no extra memory.

*)
(* standard deviation is simply the square root of the variance *)

array_sdv := SQRT(array_var(pt, size));

(* revision history
hm 1.4.2007	rev 1.0
	function created
*)
END_FUNCTION

(* POU mathematical/array functions/array_var, ST *)
FUNCTION array_var : REAL
VAR_INPUT
	pt : POINTER TO ARRAY[0..32000] OF REAL;
	size : INT;
END_VAR
VAR
	avg : REAL;
	i: INT;
	stop: INT;
END_VAR

(*
version 1.0	1 apr 2007
programmer 	hugo
tested by		tobias

this function will calculate the variance of a given array.
the function needs to be called:	array_var(adr("array"),sizeof("array"));
because this function works with pointers its very time efficient and it needs no extra memory.

*)
(* at first we calualte the arithmetic average of the array *)

stop := (size -SIZEOF(pt)) / SIZEOF(pt);
avg := pt^[0];
FOR i := 1 TO stop DO
	avg := avg + pt^[i];
END_FOR;
avg := avg / (stop + 1);

(* in a second run we calculate the variance of the array *)

array_var := EXPT(pt^[0] - avg, 2);
FOR i := 1 TO stop DO
	array_var := array_var + EXPT(pt^[i] - avg, 2);
END_FOR;
array_var := array_var / stop;

(* revision history
hm 1.4.2007	rev 1.0
	function created
*)
END_FUNCTION

(* POU mathematical/array functions/array_spr, ST *)
FUNCTION array_spr : REAL
VAR_INPUT
	pt : POINTER TO ARRAY[0..32000] OF REAL;
	size : INT;
END_VAR
VAR
	i: INT;
	stop: INT;
	array_max : REAL;
	array_min : REAL;
END_VAR

(*
version 1.0	2 oct 2006
programmer 	hugo
tested by		tobias

this function will calculate the spread of a given array.
the function needs to be called:	array_spr(adr("array"),sizeof("array"));
for example: spread of [12,0,4,1,7] is 12 - 0 = 12.
because this function works with pointers its very time efficient and it needs no extra memory.

*)
stop := (size -SIZEOF(pt)) / SIZEOF(pt);
array_min := pt^[0];
array_max := pt^[0];
FOR i := 1 TO stop DO
	IF pt^[i] > array_max THEN array_max := pt^[i];
	ELSIF pt^[i] < array_min THEN array_min := pt^[i];
	END_IF;
END_FOR;
array_spr := array_max - array_min;
END_FUNCTION

(* POU mathematical/array functions/array_sum, ST *)
FUNCTION array_sum : REAL
VAR_INPUT
	pt : POINTER TO ARRAY[0..32000] OF REAL;
	size : INT;
END_VAR
VAR
	i: INT;
	stop: INT;
END_VAR


(*
version 1.0	2 oct 2006
programmer 	hugo
tested by		tobias

this function will calculate the sum of a given array.
the function needs to be called:	array_sum(adr("array"),sizeof("array"));
because this function works with pointers its very time efficient and it needs no extra memory.

*)
stop := (size -SIZEOF(pt)) / SIZEOF(pt);
array_sum := pt^[0];
FOR i := 1 TO stop DO
	array_sum := array_sum + pt^[i];
END_FOR;
END_FUNCTION

(* POU mathematical/array functions/array_trend, ST *)
FUNCTION array_trend : REAL
VAR_INPUT
	pt : POINTER TO ARRAY[0..32000] OF REAL;
	size : INT;
END_VAR
VAR
	i: INT;
	stop: INT;
	x: REAL;
	y : REAL;
END_VAR

(*
version 1.0	2 oct 2006
programmer 	hugo
tested by		tobias

this function will calculate the trend of a given array.
trend will calculate the avg of the first half of the array and then the avg of the second half, trend = avg2 - avg1.
for example:  [0,1,4,5,3,4,6,3] = 4 - 2.5 = 1.5
the function needs to be called:	array_trend(adr("array"),sizeof("array"));
because this function works with pointers its very time efficient and it needs no extra memory.

*)
stop := (size - SIZEOF(pt)) / SIZEOF(pt);
FOR i := 0 TO stop / 2 DO x := x + pt^[i]; END_FOR;
X := x / (TRUNC(stop / 2) + 1);
IF even(stop) THEN
	FOR i := stop / 2 TO stop DO y := y + pt^[i]; END_FOR;
	y := y / (stop / 2 + 1);
ELSE
	FOR i := TRUNC(stop / 2) + 1 TO stop DO y := y + pt^[i]; END_FOR;
	y := y / (TRUNC(stop / 2) + 1);
END_IF;
array_trend := y - x;
END_FUNCTION

(* POU mathematical/functions/F_lin, ST *)
FUNCTION F_lin : REAL
VAR_INPUT
	X : REAL;
	A : REAL;
	B : REAL;
END_VAR
VAR
END_VAR

(*
version 1.0	1 sep 2006
programmer 	hugo
tested by		tobias

this function calculates the linear equation f_lin = a*x + b

*)
F_lin := A * X + B;
END_FUNCTION

(* POU mathematical/functions/F_Lin2, ST *)
FUNCTION F_Lin2 : REAL
VAR_INPUT
	X : REAL;
	X1: REAL;
	Y1 : REAL;
	X2 : REAL;
	Y2 : REAL;
END_VAR
VAR

END_VAR

(*
version 1.0	1 jan 2007
programmer 	hugo
tested by		tobias

this function calculates the linear equation f_lin = a*x + b given by two points x1/y1 and x2/y2.

*)
F_Lin2 := (Y2 - Y1) / (X2 - X1) * X + (Y1 * X1 - Y2 * X1) / (X2 - X1) + Y1;
END_FUNCTION

(* POU mathematical/functions/F_power, ST *)
FUNCTION F_power : REAL
VAR_INPUT
	a : REAL;
	x : REAL;
	n : REAL;
END_VAR
VAR
END_VAR

(*
version 1.0	1 sep 2006
programmer 	hugo
tested by		tobias

this function calculates the power equation f_power = a*x^n

*)
f_power := a * EXPT(X,N);
END_FUNCTION

(* POU mathematical/functions/F_quad, ST *)
FUNCTION F_quad : REAL
VAR_INPUT
	X : REAL;
	A : REAL;
	B : REAL;
	C : REAL;
END_VAR
VAR
END_VAR

(*
version 1.0	1 sep 2006
programmer 	hugo
tested by		tobias

this function calculates the quadratic equation f_lin = a*x + b

*)
F_quad := a * X * X + B * X + C;
END_FUNCTION

(* POU mathematical/functions/FT_avg, ST *)
FUNCTION_BLOCK FT_avg
VAR_INPUT
	in : REAL;
	en : BOOL;
	N : INT;
	rst : BOOL;
END_VAR
VAR_OUTPUT
	avg : REAL;
END_VAR
VAR
	buff : delay;
	i: INT;
	init : BOOL;
END_VAR

(*
version 1.1	7 jan 2007
programmer 	hugo
tested by		tobias

this function calculates the average over n samples from a sequential input
the input values are shifted into an N deep buffer and the avg of this buffer is diplayed at anytime on the output.
a rst will load the buffer with the current in value..

*)
(* limit n to a max of 32 because delay can do max 32 cycles *)
IF N > 32 THEN
	buff.n := 32;
ELSIF N < 0 THEN
	Buff.n := 0;
ELSE
	buff.n := N;
END_IF;

IF NOT init THEN
	FOR i := 1 TO N DO
		buff(in := in);
	END_FOR;
	avg := in;
	init := TRUE;
ELSIF rst THEN
	FOR i := 1 TO N DO
		buff(in := in);
	END_FOR;
	avg := in;
ELSIF en THEN
	buff(in := in);
	avg := avg + (in - buff.out)/N;
END_IF;

(* revision history

hm	7.1.2007	rev 1.1
	chaged rst logic to load the buffer with the actual input value instead of 0.
	added en input to allow better control of signal flow
	added init to load the buffer with in at startup to avoid rampup at beginning.
	deleted unused variable cnt.
*)
END_FUNCTION_BLOCK

(* POU mathematical/functions/FT_min_max, ST *)
FUNCTION_BLOCK FT_min_max
VAR_INPUT
	in : REAL;
	rst : BOOL;
END_VAR
VAR_OUTPUT
	mx : REAL;
	mn : REAL;
END_VAR
VAR
	init: BOOL;
END_VAR

(*
version 1.0	1 sep 2006
programmer 	hugo
tested by		tobias

this function block stores the min and max value of an input signal.
when rst is true the mn and mx outputs are set to the in value.
when a rst is never active the function autoresets to the in value at startup.
since the input might not be present at first cycle the mn and mx are set during second cycle.

*)
IF rst OR NOT init THEN
	mn := in;
	mx := in;
	init := 1;
ELSIF in < mn THEN mn := in;
ELSIF in > mx THEN mx := in;
END_IF;
END_FUNCTION_BLOCK

(* POU mathematical/functions/POLYNOM_INT, ST *)
FUNCTION POLYNOM_INT : REAL
VAR_INPUT
	X : REAL;
	XY : ARRAY[1..5,0..1] OF REAL;
	Pts : INT;
END_VAR
VAR
	I, J : INT;
	init: BOOL;
END_VAR

(*
	version 1.0	7 oct 2007
	programmer 	oscat
	tested BY		oscat

POLYNOM_INT calculates an output based on a Polynom interpolation of up to 5 coordinates given in an array
the indut coordinates have to start at the lowest array position and must be sorted ba ascending X values.

*)
(*make sure n is bound within the array size *)
IF pts > 5 THEN pts := 5; END_IF;

(* this part is only to calculate the polynom parameters, which are then stores in the Y array
	the array values, it is not needed during runtime, unless the parameters will change during runtime
	the remaining code without this setup code can be used within a function to calculate specific functions
	the content of the arrays is then used as constant values within the function *)
IF NOT init THEN
	init := TRUE;
	FOR i := 1 TO pts DO
       	FOR j := pts TO i + 1 BY -1 DO
           		XY[j,1] := (XY[j,1] - XY[j-1,1]) / (XY[j,0] - XY[j-i,0]);
		END_FOR;
	END_FOR;
END_IF;

(* this part is the actual calculation *)
POLYNOM_INT := 0;
FOR i := pts TO 1 BY -1DO
       POLYNOM_INT := POLYNOM_INT * (X - XY[i,0]) + XY[i,1];
END_FOR;


(* revision history
hm		8. okt 2007	rev 1.0
	original version

*)
END_FUNCTION

(* POU mathematical/Geometry/circle_A, ST *)
FUNCTION circle_A : REAL
VAR_INPUT
	rx : REAL;
	ax : REAL;
END_VAR
VAR
END_VAR

(*
version 1.0	16 oct 2007
programmer 	hugo
tested by		tobias

circle_A calculates the Area of a circle segement if ax = 360 the whole circle is calculated


*)
circle_A := PI1 * EXPT(Rx,2) / 360 * Ax;

(* revision histroy
hm	16. oct 2007	rev 1.0
	original version

*)
END_FUNCTION

(* POU mathematical/Geometry/circle_C, ST *)
FUNCTION circle_C : REAL
VAR_INPUT
	Rx : REAL;
	Ax : REAL;
END_VAR
VAR
END_VAR

(*
version 1.0	16 oct 2007
programmer 	hugo
tested by		tobias

circle_C calculates the Circumference of a circle  if ax = 360 the whole circle is calculated

*)
circle_C := PI2 * Rx * Ax / 360;

(* revision histroy
hm	16. oct 2007	rev 1.0
	original version

*)
END_FUNCTION

(* POU mathematical/Geometry/cone_V, ST *)
FUNCTION cone_V : REAL
VAR_INPUT
	rx : REAL;
	hx : REAL;
END_VAR
VAR
END_VAR

(*
version 1.0	17 oct 2007
programmer 	hugo
tested by		tobias

cone_V calculates the Volume of a cone

*)
cone_V := PI1 / 3 * EXPT(Rx,2) * hx;

(* revision histroy
hm	17. oct 2007	rev 1.0
	original version

*)
END_FUNCTION

(* POU mathematical/Geometry/ellipse_A, ST *)
FUNCTION ellipse_A : REAL
VAR_INPUT
	R1 : REAL;
	R2 : REAL;
END_VAR
VAR
END_VAR

(*
version 1.0	16 oct 2007
programmer 	hugo
tested by		tobias

ellipse_A calculates the Area of an ellipe based on the two radians R1 and R2


*)
ellipse_A := PI1 * R1 * R2;

(* revision histroy
hm	16. oct 2007	rev 1.0
	original version

*)
END_FUNCTION

(* POU mathematical/Geometry/ellipse_C, ST *)
FUNCTION ellipse_C : REAL
VAR_INPUT
	R1 : REAL;
	R2 : REAL;
END_VAR
VAR
END_VAR

(*
version 1.0	16 oct 2007
programmer 	hugo
tested by		tobias

ellipse_C calculates the circumference of an ellipe based on the two radians R1 and R2

*)
ellipse_C := PI1 * (3*(R1+R2) - SQRT((3*r1 + R2)*(3*r2 + r1)));

(* revision histroy
hm	16. oct 2007	rev 1.0
	original version

*)
END_FUNCTION

(* POU mathematical/Geometry/sphere_V, ST *)
FUNCTION sphere_V : REAL
VAR_INPUT
	rx : REAL;
END_VAR
VAR
END_VAR

(*
version 1.0	16 oct 2007
programmer 	hugo
tested by		tobias

sphere_V calculates the Volume of a Sphere


*)
sphere_V := 4 / 3 * PI1 * EXPT(Rx,3);

(* revision histroy
hm	16. oct 2007	rev 1.0
	original version

*)
END_FUNCTION

(* POU mathematical/Geometry/triangle_A, ST *)
FUNCTION triangle_A : REAL
VAR_INPUT
	S1 : REAL;
	A : REAL;
	S2 : REAL;
	S3 : REAL;
END_VAR
VAR
END_VAR

(*
version 1.0	16 oct 2007
programmer 	hugo
tested by		tobias

triangle_A calculates the Area of a triangle.
if any input is 0 it will be neglected and the are will be calculated from eiter:
two sides and an angle (s1 and S2 and the angle A1) or 3 sides.


*)
IF A = 0 THEN
	triangle_A := SQRT((S1+S2+S3) * (S1+S2-S3) * (S2+S3-S1) * (S3+S1-S2)) / 4;
ELSE
	triangle_A := S1 * S2 * SIN(Rad(A)) / 2;
END_IF;
(* revision histroy
hm	16. oct 2007	rev 1.0
	original version

*)
END_FUNCTION

(* POU mathematical/acosH, ST *)
FUNCTION acosH : REAL
VAR_INPUT
	X : REAL;
END_VAR
VAR
END_VAR


(*
version 1.0	12 jan 2007
programmer 	hugo
tested by		tobias

this function calculates the arcus cos hyperbolicus

*)
acosH := LN(X + SQRT(EXPT(x,2)-1));
END_FUNCTION

(* POU mathematical/acotH, ST *)
FUNCTION acotH : REAL
VAR_INPUT
	X : REAL;
END_VAR
VAR
END_VAR


(*
version 1.0	12 jan 2007
programmer 	hugo
tested by		tobias

this function calculates the arcus cotangens hyperbolicus

*)
acotH := LN((x+1)/(x-1))/2;
END_FUNCTION

(* POU mathematical/asinH, ST *)
FUNCTION asinH : REAL
VAR_INPUT
	X : REAL;
END_VAR
VAR
END_VAR


(*
version 1.0	12 jan 2007
programmer 	hugo
tested by		tobias

this function calculates the arcus sin hyperbolicus

*)
asinH := LN(X + SQRT(EXPT(x,2)+1));
END_FUNCTION

(* POU mathematical/atanH, ST *)
FUNCTION atanH : REAL
VAR_INPUT
	X : REAL;
END_VAR
VAR
END_VAR


(*
version 1.0	12 jan 2007
programmer 	hugo
tested by		tobias

this function calculates the arcus tangens hyperbolicus

*)
atanH := LN((1+x)/(1-x)) / 2;
END_FUNCTION

(* POU mathematical/ceil, ST *)
FUNCTION ceil : INT
VAR_INPUT
	X : REAL;
END_VAR
VAR
END_VAR


(*
version 1.0	7 feb 2007
programmer 	hugo
tested by		tobias

This is a rounding function which returns the smallest possible integer which is greater or equal to X.
ceil(3.14) = 4
ceil(-3.14) = -3

*)
ceil := TRUNC(X);
IF ceil < X THEN
	ceil := ceil + 1;
END_IF;
END_FUNCTION

(* POU mathematical/cosH, ST *)
FUNCTION cosH : REAL
VAR_INPUT
	X : REAL;
END_VAR
VAR
END_VAR


(*
version 1.0	12 jan 2007
programmer 	hugo
tested by		tobias

this function calculates the cos hyperbolicus

*)
cosH := (EXPT(e,x) + EXPT(e,-x))/2;
END_FUNCTION

(* POU mathematical/cotH, ST *)
FUNCTION cotH : REAL
VAR_INPUT
	X : REAL;
END_VAR
VAR
END_VAR


(*
version 1.0	12 jan 2007
programmer 	hugo
tested by		tobias

this function calculates the cotangens hyperbolicus

*)
cotH := (EXPT(e, 2 * x) + 1) / (EXPT(e, 2 * x) - 1);
END_FUNCTION

(* POU mathematical/fact, ST *)
FUNCTION fact : INT
VAR_INPUT
	X : INT;
END_VAR
VAR
	i: INT;
END_VAR

(*
version 1.1	4 mar 2007
programmer 	hugo
tested by		tobias

this function calculates the factorial of x
this simple factorial only calculates factorials for inputs up to 7
if the input is negative or higher then 7 the output will be -1.

*)
IF x >= 0 AND x < 8 THEN
	fact := 1;
	i := 1;
	WHILE i <= x DO
		fact := fact * i;
		i := i + 1;
	END_WHILE;
ELSE
	fact := -1;
END_IF;

(* revision history
hm 4.3.2007	rev 1.1
	changed a critical error where while loop was indefinite.

*)
END_FUNCTION

(* POU mathematical/floor, ST *)
FUNCTION floor : INT
VAR_INPUT
	X : REAL;
END_VAR
VAR
END_VAR


(*
version 1.0	7 feb 2007
programmer 	hugo
tested by		tobias

This is a rounding function which returns the biggest possible integer which is less or equal to X.
floor(3.14) = 3
floor(-3.14) = -4

*)
floor := TRUNC(X);
IF floor > X THEN
	floor := floor - 1;
END_IF;
END_FUNCTION

(* POU mathematical/inc, ST *)
FUNCTION inc : INT
VAR_INPUT
	X : INT;
	D : INT;
	M : INT;
END_VAR
VAR
END_VAR


(*
version 1.0	7 feb 2007
programmer 	hugo
tested by		tobias

This is a increment function which increments the input X by the value D and compares the result with M.
if the output exceeds M it will continue to count from 0 again.

*)
inc := (X + D) MOD (m+1);
END_FUNCTION

(* POU mathematical/max3, ST *)
FUNCTION max3 : REAL
VAR_INPUT
	in1 : REAL;
	in2 : REAL;
	in3 : REAL;
END_VAR
VAR
END_VAR

(*
version 1.0	1 jan 2007
programmer 	hugo
tested by		tobias

this function returns the highest of 3 real values

*)
IF in1 >= in2 AND in1 >= in3 THEN
	max3 := in1;
ELSIF in2 >= in1 AND in2 >= in3 THEN
	max3 := in2;
ELSE
	max3 := in3;
END_IF;
END_FUNCTION

(* POU mathematical/min3, ST *)
FUNCTION min3 : REAL
VAR_INPUT
	in1 : REAL;
	in2 : REAL;
	in3 : REAL;
END_VAR
VAR
END_VAR

(*
version 1.0	1 jan 2007
programmer 	hugo
tested by		tobias

this function returns the lowest of 3 real values

*)
IF in1 <= in2 AND in1 <= in3 THEN
	min3 := in1;
ELSIF in2 <= in1 AND in2 <= in3 THEN
	min3 := in2;
ELSE
	min3 := in3;
END_IF;
END_FUNCTION

(* POU mathematical/MUL_ADD, ST *)
FUNCTION MUL_ADD : REAL
VAR_INPUT
	X : REAL;
	K : REAL;
	O : REAL;
END_VAR
VAR
END_VAR

(*
version 1.1	11 nov 2007
programmer 	hugo
tested by		tobias

this function multiplies an input X with K and adds Offset O to the result.

*)
MUL_ADD := X * K + O;

(* revision history
hm	28. feb 2007
	original version

hm	11.nov 2007		rev 1.1
	deleted preset values for K and O this makes no sense for a function

*)
END_FUNCTION

(* POU mathematical/neg, ST *)
FUNCTION neg : INT
VAR_INPUT
	in : INT;
END_VAR
VAR
	X : WORD := 2#1111_1111_1111_1111;
END_VAR

(*
version 1.0	11 nov 2007
programmer 	hugo
tested by		tobias

this function return the value of in multiplied by -1

*)
neg := WORD_TO_INT(INT_TO_WORD(in - 1) XOR X);

(* revision history
hm 11.11.2007	rev 1.0
	original version

*)
END_FUNCTION

(* POU mathematical/round, ST *)
FUNCTION round : REAL
VAR_INPUT
	in : REAL;
	N : INT;
END_VAR
VAR
END_VAR

(*
version 1.0	1 sep 2006
programmer 	hugo
tested by		tobias

this function rounds a real down to n digits behind the comma.
round(3.1415,1) = 3.1

*)
round := TRUNC(in * EXPT(10,N) + 0.5)/EXPT(10,N);
END_FUNCTION

(* POU mathematical/sign_I, ST *)
FUNCTION sign_I : BOOL
VAR_INPUT
	in : INT;
END_VAR
VAR
END_VAR

(*
version 1.1	3 mar 2007
programmer 	hugo
tested by		tobias

this function return true if the integer input is negative

*)
IF in < 0 THEN
	sign_I := TRUE;
ELSE
	sign_I := FALSE;
END_IF;

(* revision history
hm 3.3.2007	rev 1.1
	changed method of function for better compatibility to other systems

*)
END_FUNCTION

(* POU mathematical/sinH, ST *)
FUNCTION sinH : REAL
VAR_INPUT
	X : REAL;
END_VAR
VAR
END_VAR


(*
version 1.0	12 jan 2007
programmer 	hugo
tested by		tobias

this function calculates the sin hyperbolicus

*)
sinH := (EXPT(e,x) - EXPT(e,-x))/2;
END_FUNCTION

(* POU mathematical/sqrtn, ST *)
FUNCTION sqrtn : REAL
VAR_INPUT
	X : REAL;
	N : INT;
END_VAR
VAR
END_VAR

(*
version 1.0	12 jan 2007
programmer 	hugo
tested by		tobias

this function calculates the nth root function of X according to the formula sqrtn = x^(1/n).

*)
IF N > 1 THEN
	sqrtn := EXPT(x, 1.0 / INT_TO_REAL(n));
END_IF;
END_FUNCTION

(* POU mathematical/tanH, ST *)
FUNCTION tanH : REAL
VAR_INPUT
	X : REAL;
END_VAR
VAR
END_VAR


(*
version 1.0	12 jan 2007
programmer 	hugo
tested by		tobias

this function calculates the tangens hyperbolicus

*)
tanH := -2 / (EXPT(e, -2 * x) + 1) + 1;
END_FUNCTION

(* POU mathematical/window, ST *)
FUNCTION window : BOOL
VAR_INPUT
	low : REAL;
	in : REAL;
	high : REAL;
END_VAR
VAR
END_VAR

(*
	version 1.1	22 jan 2007
	programmer 	hugo
	tested BY		tobias

this checks a signal if the signal is between the upper and lower limit
*)
window := in < high AND in > low;


(* revision history
hm	22.1.2007	rev 1.1
	changed the order of inputs to low, in, high

*)
END_FUNCTION

(* POU mathematical/window2, ST *)
FUNCTION window2 : BOOL
VAR_INPUT
	low : REAL;
	in : REAL;
	high : REAL;
END_VAR
VAR
END_VAR

(*
	version 1.0	31 oct 2007
	programmer 	hugo
	tested BY		tobias

this checks a signal if the signal is between the upper and lower limit including the two limits
*)
window2 := in <= high AND in >= low;


(* revision history
hm	31.10.2007	rev 1.0
	original version

*)
END_FUNCTION

